// TIA Portal project "EbAndon v2_0_1" (V15)

(* hardware
DEVICE "S71500/ET200MP station_1"  S7-1500 station
   slot 0: "Rail_0"  Rack  6ES7 590-1***0-0AA0
   slot 1: "PLC_1"  CPU 1515F-2 PN  6ES7 515-2FM01-0AB0  V2.5
      slot 3: "CPU display_1"  6ES7591-1BA00-0AA0
DEVICE "HMI_1"  TP1500 Comfort PRO
   slot 0: "HMI_1"  TP1500 Comfort PRO  6AV2 124-0QC24-1AX0  15.0.0.0
   slot 1: "HMI_RT_1"  TP1500 Comfort PRO  6AV2 124-0QC24-1AX0  15.0.0.0
   slot 5: "HMI_1.IE_CP_1"  PROFINET Interface  15.0.0.0
      slot 1: "PROFINET Interface_1"  PROFINET Interface
         slot 1: "Port_1"  Port
         slot 2: "Port_2"  Port
   slot 6: "HMI_1.IE_CP_2"  PROFINET Interface  15.0.0.0
      slot 1: "PROFINET Interface_GBit"  PROFINET Interface
         slot 1: "Port_1"  Port
   slot 7: "HMI_1.MPI/DP_CP_1"  MPI/DP Interface  15.0.0.0
DEVICE "ET 200SP station_1"  ET 200SP-Station
   slot 0: "Rack_0"  Rack  6ES5 710-8MAx1
   slot 0: "station6et200sp"  IM 155-6 PN ST  6ES7 155-6AU01-0BN0  V4.1
   slot 1: "DQ 8x24VDC/0.5A ST_1"  DQ 8x24VDC/0.5A ST  6ES7 132-6BF01-0BA0  V0.0
      slot 1: "DQ 8x24VDC/0.5A ST_1"  DQ 8x24VDC/0.5A ST
   slot 2: "DQ 8x24VDC/0.5A ST_2"  DQ 8x24VDC/0.5A ST  6ES7 132-6BF01-0BA0  V0.0
      slot 1: "DQ 8x24VDC/0.5A ST_2"  DQ 8x24VDC/0.5A ST
   slot 3: "DQ 8x24VDC/0.5A ST_3"  DQ 8x24VDC/0.5A ST  6ES7 132-6BF01-0BA0  V0.0
      slot 1: "DQ 8x24VDC/0.5A ST_3"  DQ 8x24VDC/0.5A ST
   slot 4: "Server module_1"  Server module  6ES7 193-6PA00-0AA0  V1.1
      slot 1: "Server module_1"  Server module
   slot 127: "BA 2xRJ45"  BA 2xRJ45  6ES7 193-6AR00-0AA0  V0.0
      slot 1: "Port_1"  6ES7 193-6AR00-0AA0  V0.0
      slot 2: "Port_2"  6ES7 193-6AR00-0AA0  V0.0
DEVICE "ET 200SP station_2"  ET 200SP-Station
   slot 0: "Rack_0"  Rack  6ES5 710-8MAx1
   slot 0: "station7et200sp"  IM 155-6 PN ST  6ES7 155-6AU01-0BN0  V4.1
   slot 1: "DQ 8x24VDC/0.5A ST_1"  DQ 8x24VDC/0.5A ST  6ES7 132-6BF01-0BA0  V0.0
      slot 1: "DQ 8x24VDC/0.5A ST_1"  DQ 8x24VDC/0.5A ST
   slot 2: "DQ 8x24VDC/0.5A ST_2"  DQ 8x24VDC/0.5A ST  6ES7 132-6BF01-0BA0  V0.0
      slot 1: "DQ 8x24VDC/0.5A ST_2"  DQ 8x24VDC/0.5A ST
   slot 3: "DQ 8x24VDC/0.5A ST_3"  DQ 8x24VDC/0.5A ST  6ES7 132-6BF01-0BA0  V0.0
      slot 1: "DQ 8x24VDC/0.5A ST_3"  DQ 8x24VDC/0.5A ST
   slot 4: "Server module_1"  Server module  6ES7 193-6PA00-0AA0  V1.1
      slot 1: "Server module_1"  Server module
   slot 127: "BA 2xRJ45"  BA 2xRJ45  6ES7 193-6AR00-0AA0  V0.0
      slot 1: "Port_1"  6ES7 193-6AR00-0AA0  V0.0
      slot 2: "Port_2"  6ES7 193-6AR00-0AA0  V0.0
DEVICE "ET 200SP station_3"  ET 200SP-Station
   slot 0: "Rack_0"  Rack  6ES5 710-8MAx1
   slot 0: "station8et200sp"  IM 155-6 PN ST  6ES7 155-6AU01-0BN0  V4.1
   slot 1: "DQ 8x24VDC/0.5A ST_1"  DQ 8x24VDC/0.5A ST  6ES7 132-6BF01-0BA0  V0.0
      slot 1: "DQ 8x24VDC/0.5A ST_1"  DQ 8x24VDC/0.5A ST
   slot 2: "DQ 8x24VDC/0.5A ST_2"  DQ 8x24VDC/0.5A ST  6ES7 132-6BF01-0BA0  V0.0
      slot 1: "DQ 8x24VDC/0.5A ST_2"  DQ 8x24VDC/0.5A ST
   slot 3: "DQ 8x24VDC/0.5A ST_3"  DQ 8x24VDC/0.5A ST  6ES7 132-6BF01-0BA0  V0.0
      slot 1: "DQ 8x24VDC/0.5A ST_3"  DQ 8x24VDC/0.5A ST
   slot 4: "Server module_1"  Server module  6ES7 193-6PA00-0AA0  V1.1
      slot 1: "Server module_1"  Server module
   slot 127: "BA 2xRJ45"  BA 2xRJ45  6ES7 193-6AR00-0AA0  V0.0
      slot 1: "Port_1"  6ES7 193-6AR00-0AA0  V0.0
      slot 2: "Port_2"  6ES7 193-6AR00-0AA0  V0.0
DEVICE "KP8_1"  SIMATIC Key Panel
   slot 0: "Rack"  Rail  V1.0
   slot 0: "station8kp8"  KP8  6AV3 688-3AY36-0AX0  R01.00.00
DEVICE "KP8_2"  SIMATIC Key Panel
   slot 0: "Rack"  Rail  V1.0
   slot 0: "station7kp8"  KP8  6AV3 688-3AY36-0AX0  R01.00.00
DEVICE "KP8_3"  SIMATIC Key Panel
   slot 0: "Rack"  Rail  V1.0
   slot 0: "station6kp8"  KP8  6AV3 688-3AY36-0AX0  R01.00.00
DEVICE "KP8_4"  SIMATIC Key Panel
   slot 0: "Rack"  Rail  V1.0
   slot 0: "station9kp8"  KP8  6AV3 688-3AY36-0AX0  R01.00.00
DEVICE "ET 200SP station_4"  ET 200SP-Station
   slot 0: "Rack_0"  Rack  6ES5 710-8MAx1
   slot 0: "station9et200sp"  IM 155-6 PN ST  6ES7 155-6AU01-0BN0  V4.1
   slot 1: "DQ 8x24VDC/0.5A ST_1"  DQ 8x24VDC/0.5A ST  6ES7 132-6BF01-0BA0  V0.0
      slot 1: "DQ 8x24VDC/0.5A ST_1"  DQ 8x24VDC/0.5A ST
   slot 2: "DQ 8x24VDC/0.5A ST_2"  DQ 8x24VDC/0.5A ST  6ES7 132-6BF01-0BA0  V0.0
      slot 1: "DQ 8x24VDC/0.5A ST_2"  DQ 8x24VDC/0.5A ST
   slot 3: "DQ 8x24VDC/0.5A ST_3"  DQ 8x24VDC/0.5A ST  6ES7 132-6BF01-0BA0  V0.0
      slot 1: "DQ 8x24VDC/0.5A ST_3"  DQ 8x24VDC/0.5A ST
   slot 4: "Server module_1"  Server module  6ES7 193-6PA00-0AA0  V1.1
      slot 1: "Server module_1"  Server module
   slot 127: "BA 2xRJ45"  BA 2xRJ45  6ES7 193-6AR00-0AA0  V0.0
      slot 1: "Port_1"  6ES7 193-6AR00-0AA0  V0.0
      slot 2: "Port_2"  6ES7 193-6AR00-0AA0  V0.0
DEVICE "ET 200SP station_5"  ET 200SP-Station
   slot 0: "Rack_0"  Rack  6ES5 710-8MAx1
   slot 0: "station10et200sp"  IM 155-6 PN ST  6ES7 155-6AU01-0BN0  V4.1
   slot 1: "DQ 8x24VDC/0.5A ST_1"  DQ 8x24VDC/0.5A ST  6ES7 132-6BF01-0BA0  V0.0
      slot 1: "DQ 8x24VDC/0.5A ST_1"  DQ 8x24VDC/0.5A ST
   slot 2: "DQ 8x24VDC/0.5A ST_2"  DQ 8x24VDC/0.5A ST  6ES7 132-6BF01-0BA0  V0.0
      slot 1: "DQ 8x24VDC/0.5A ST_2"  DQ 8x24VDC/0.5A ST
   slot 3: "DQ 8x24VDC/0.5A ST_3"  DQ 8x24VDC/0.5A ST  6ES7 132-6BF01-0BA0  V0.0
      slot 1: "DQ 8x24VDC/0.5A ST_3"  DQ 8x24VDC/0.5A ST
   slot 4: "Server module_1"  Server module  6ES7 193-6PA00-0AA0  V1.1
      slot 1: "Server module_1"  Server module
   slot 127: "BA 2xRJ45"  BA 2xRJ45  6ES7 193-6AR00-0AA0  V0.0
      slot 1: "Port_1"  6ES7 193-6AR00-0AA0  V0.0
      slot 2: "Port_2"  6ES7 193-6AR00-0AA0  V0.0
DEVICE "KP8_5"  SIMATIC Key Panel
   slot 0: "Rack"  Rail  V1.0
   slot 0: "station10kp8"  KP8  6AV3 688-3AY36-0AX0  R01.00.00
DEVICE "KP8_6"  SIMATIC Key Panel
   slot 0: "Rack"  Rail  V1.0
   slot 0: "station11kp8"  KP8  6AV3 688-3AY36-0AX0  R01.00.00
DEVICE "ET 200SP station_6"  ET 200SP-Station
   slot 0: "Rack_0"  Rack  6ES5 710-8MAx1
   slot 0: "station11et200sp"  IM 155-6 PN ST  6ES7 155-6AU01-0BN0  V4.1
   slot 1: "DQ 8x24VDC/0.5A ST_1"  DQ 8x24VDC/0.5A ST  6ES7 132-6BF01-0BA0  V0.0
      slot 1: "DQ 8x24VDC/0.5A ST_1"  DQ 8x24VDC/0.5A ST
   slot 2: "DQ 8x24VDC/0.5A ST_2"  DQ 8x24VDC/0.5A ST  6ES7 132-6BF01-0BA0  V0.0
      slot 1: "DQ 8x24VDC/0.5A ST_2"  DQ 8x24VDC/0.5A ST
   slot 3: "DQ 8x24VDC/0.5A ST_3"  DQ 8x24VDC/0.5A ST  6ES7 132-6BF01-0BA0  V0.0
      slot 1: "DQ 8x24VDC/0.5A ST_3"  DQ 8x24VDC/0.5A ST
   slot 4: "Server module_1"  Server module  6ES7 193-6PA00-0AA0  V1.1
      slot 1: "Server module_1"  Server module
   slot 127: "BA 2xRJ45"  BA 2xRJ45  6ES7 193-6AR00-0AA0  V0.0
      slot 1: "Port_1"  6ES7 193-6AR00-0AA0  V0.0
      slot 2: "Port_2"  6ES7 193-6AR00-0AA0  V0.0
DEVICE "KP8_7"  SIMATIC Key Panel
   slot 0: "Rack"  Rail  V1.0
   slot 0: "station01kp8"  KP8  6AV3 688-3AY36-0AX0  R01.00.00
DEVICE "ET 200SP station_7"  ET 200SP-Station
   slot 0: "Rack_0"  Rack  6ES5 710-8MAx1
   slot 0: "station01et200sp"  IM 155-6 PN ST  6ES7 155-6AU01-0BN0  V4.1
   slot 1: "DQ 8x24VDC/0.5A ST_1"  DQ 8x24VDC/0.5A ST  6ES7 132-6BF01-0BA0  V0.0
      slot 1: "DQ 8x24VDC/0.5A ST_1"  DQ 8x24VDC/0.5A ST
   slot 2: "DQ 8x24VDC/0.5A ST_2"  DQ 8x24VDC/0.5A ST  6ES7 132-6BF01-0BA0  V0.0
      slot 1: "DQ 8x24VDC/0.5A ST_2"  DQ 8x24VDC/0.5A ST
   slot 3: "DQ 8x24VDC/0.5A ST_3"  DQ 8x24VDC/0.5A ST  6ES7 132-6BF01-0BA0  V0.0
      slot 1: "DQ 8x24VDC/0.5A ST_3"  DQ 8x24VDC/0.5A ST
   slot 4: "Server module_1"  Server module  6ES7 193-6PA00-0AA0  V1.1
      slot 1: "Server module_1"  Server module
   slot 127: "BA 2xRJ45"  BA 2xRJ45  6ES7 193-6AR00-0AA0  V0.0
      slot 1: "Port_1"  6ES7 193-6AR00-0AA0  V0.0
      slot 2: "Port_2"  6ES7 193-6AR00-0AA0  V0.0
DEVICE "ET 200SP station_8"  ET 200SP-Station
   slot 0: "Rack_0"  Rack  6ES5 710-8MAx1
   slot 0: "station02et200sp"  IM 155-6 PN ST  6ES7 155-6AU01-0BN0  V4.1
   slot 1: "DQ 8x24VDC/0.5A ST_1"  DQ 8x24VDC/0.5A ST  6ES7 132-6BF01-0BA0  V0.0
      slot 1: "DQ 8x24VDC/0.5A ST_1"  DQ 8x24VDC/0.5A ST
   slot 2: "DQ 8x24VDC/0.5A ST_2"  DQ 8x24VDC/0.5A ST  6ES7 132-6BF01-0BA0  V0.0
      slot 1: "DQ 8x24VDC/0.5A ST_2"  DQ 8x24VDC/0.5A ST
   slot 3: "DQ 8x24VDC/0.5A ST_3"  DQ 8x24VDC/0.5A ST  6ES7 132-6BF01-0BA0  V0.0
      slot 1: "DQ 8x24VDC/0.5A ST_3"  DQ 8x24VDC/0.5A ST
   slot 4: "Server module_1"  Server module  6ES7 193-6PA00-0AA0  V1.1
      slot 1: "Server module_1"  Server module
   slot 127: "BA 2xRJ45"  BA 2xRJ45  6ES7 193-6AR00-0AA0  V0.0
      slot 1: "Port_1"  6ES7 193-6AR00-0AA0  V0.0
      slot 2: "Port_2"  6ES7 193-6AR00-0AA0  V0.0
DEVICE "KP8_8"  SIMATIC Key Panel
   slot 0: "Rack"  Rail  V1.0
   slot 0: "station02kp8"  KP8  6AV3 688-3AY36-0AX0  R01.00.00
DEVICE "KP8_9"  SIMATIC Key Panel
   slot 0: "Rack"  Rail  V1.0
   slot 0: "station03kp8"  KP8  6AV3 688-3AY36-0AX0  R01.00.00
DEVICE "KP8_10"  SIMATIC Key Panel
   slot 0: "Rack"  Rail  V1.0
   slot 0: "station04kp8"  KP8  6AV3 688-3AY36-0AX0  R01.00.00
DEVICE "KP8_11"  SIMATIC Key Panel
   slot 0: "Rack"  Rail  V1.0
   slot 0: "station05kp8"  KP8  6AV3 688-3AY36-0AX0  R01.00.00
DEVICE "ET 200SP station_9"  ET 200SP-Station
   slot 0: "Rack_0"  Rack  6ES5 710-8MAx1
   slot 0: "station03et200sp"  IM 155-6 PN ST  6ES7 155-6AU01-0BN0  V4.1
   slot 1: "DQ 8x24VDC/0.5A ST_1"  DQ 8x24VDC/0.5A ST  6ES7 132-6BF01-0BA0  V0.0
      slot 1: "DQ 8x24VDC/0.5A ST_1"  DQ 8x24VDC/0.5A ST
   slot 2: "DQ 8x24VDC/0.5A ST_2"  DQ 8x24VDC/0.5A ST  6ES7 132-6BF01-0BA0  V0.0
      slot 1: "DQ 8x24VDC/0.5A ST_2"  DQ 8x24VDC/0.5A ST
   slot 3: "DQ 8x24VDC/0.5A ST_3"  DQ 8x24VDC/0.5A ST  6ES7 132-6BF01-0BA0  V0.0
      slot 1: "DQ 8x24VDC/0.5A ST_3"  DQ 8x24VDC/0.5A ST
   slot 4: "Server module_1"  Server module  6ES7 193-6PA00-0AA0  V1.1
      slot 1: "Server module_1"  Server module
   slot 127: "BA 2xRJ45"  BA 2xRJ45  6ES7 193-6AR00-0AA0  V0.0
      slot 1: "Port_1"  6ES7 193-6AR00-0AA0  V0.0
      slot 2: "Port_2"  6ES7 193-6AR00-0AA0  V0.0
DEVICE "ET 200SP station_10"  ET 200SP-Station
   slot 0: "Rack_0"  Rack  6ES5 710-8MAx1
   slot 0: "station04et200sp"  IM 155-6 PN ST  6ES7 155-6AU01-0BN0  V4.1
   slot 1: "DQ 8x24VDC/0.5A ST_1"  DQ 8x24VDC/0.5A ST  6ES7 132-6BF01-0BA0  V0.0
      slot 1: "DQ 8x24VDC/0.5A ST_1"  DQ 8x24VDC/0.5A ST
   slot 2: "DQ 8x24VDC/0.5A ST_2"  DQ 8x24VDC/0.5A ST  6ES7 132-6BF01-0BA0  V0.0
      slot 1: "DQ 8x24VDC/0.5A ST_2"  DQ 8x24VDC/0.5A ST
   slot 3: "DQ 8x24VDC/0.5A ST_3"  DQ 8x24VDC/0.5A ST  6ES7 132-6BF01-0BA0  V0.0
      slot 1: "DQ 8x24VDC/0.5A ST_3"  DQ 8x24VDC/0.5A ST
   slot 4: "Server module_1"  Server module  6ES7 193-6PA00-0AA0  V1.1
      slot 1: "Server module_1"  Server module
   slot 127: "BA 2xRJ45"  BA 2xRJ45  6ES7 193-6AR00-0AA0  V0.0
      slot 1: "Port_1"  6ES7 193-6AR00-0AA0  V0.0
      slot 2: "Port_2"  6ES7 193-6AR00-0AA0  V0.0
DEVICE "ET 200SP station_11"  ET 200SP-Station
   slot 0: "Rack_0"  Rack  6ES5 710-8MAx1
   slot 0: "station05et200sp"  IM 155-6 PN ST  6ES7 155-6AU01-0BN0  V4.1
   slot 1: "DQ 8x24VDC/0.5A ST_1"  DQ 8x24VDC/0.5A ST  6ES7 132-6BF01-0BA0  V0.0
      slot 1: "DQ 8x24VDC/0.5A ST_1"  DQ 8x24VDC/0.5A ST
   slot 2: "DQ 8x24VDC/0.5A ST_2"  DQ 8x24VDC/0.5A ST  6ES7 132-6BF01-0BA0  V0.0
      slot 1: "DQ 8x24VDC/0.5A ST_2"  DQ 8x24VDC/0.5A ST
   slot 3: "DQ 8x24VDC/0.5A ST_3"  DQ 8x24VDC/0.5A ST  6ES7 132-6BF01-0BA0  V0.0
      slot 1: "DQ 8x24VDC/0.5A ST_3"  DQ 8x24VDC/0.5A ST
   slot 4: "Server module_1"  Server module  6ES7 193-6PA00-0AA0  V1.1
      slot 1: "Server module_1"  Server module
   slot 127: "BA 2xRJ45"  BA 2xRJ45  6ES7 193-6AR00-0AA0  V0.0
      slot 1: "Port_1"  6ES7 193-6AR00-0AA0  V0.0
      slot 2: "Port_2"  6ES7 193-6AR00-0AA0  V0.0
DEVICE "PC-System_1"  SIMATIC PC station
   slot 0: "SIMATIC PC station"  Rail  SIMATIC PC-Station  V1.0
      slot 125: "Stationmanager"  Station_Manager  V6.0.4
   slot 1: "HMI_RT_2"  WinCC RT Advanced  6AV2 104-0xxxx-xxxx  15.0.0.0
      slot 33792: "Host interface"  Host interface
   slot 2: "IE general_1"  IE General  IE_CP  V8.2.0
DEVICE "ET 200SP station_12"  ET 200SP-Station
   slot 0: "Rack_0"  Rack  6ES5 710-8MAx1
   slot 0: "chm1et200sp"  IM 155-6 PN ST  6ES7 155-6AU01-0BN0  V4.1
   slot 1: "DQ 8x24VDC/0.5A ST_1"  DQ 8x24VDC/0.5A ST  6ES7 132-6BF01-0BA0  V0.0
      slot 1: "DQ 8x24VDC/0.5A ST_1"  DQ 8x24VDC/0.5A ST
   slot 2: "DQ 8x24VDC/0.5A ST_2"  DQ 8x24VDC/0.5A ST  6ES7 132-6BF01-0BA0  V0.0
      slot 1: "DQ 8x24VDC/0.5A ST_2"  DQ 8x24VDC/0.5A ST
   slot 3: "DQ 8x24VDC/0.5A ST_3"  DQ 8x24VDC/0.5A ST  6ES7 132-6BF01-0BA0  V0.0
      slot 1: "DQ 8x24VDC/0.5A ST_3"  DQ 8x24VDC/0.5A ST
   slot 4: "Server module_1"  Server module  6ES7 193-6PA00-0AA0  V1.1
      slot 1: "Server module_1"  Server module
   slot 127: "BA 2xRJ45"  BA 2xRJ45  6ES7 193-6AR00-0AA0  V0.0
      slot 1: "Port_1"  6ES7 193-6AR00-0AA0  V0.0
      slot 2: "Port_2"  6ES7 193-6AR00-0AA0  V0.0
DEVICE "KP8_12"  SIMATIC Key Panel
   slot 0: "Rack"  Rail  V1.0
   slot 0: "chm1kp8"  KP8  6AV3 688-3AY36-0AX0  R01.00.00
DEVICE "ET 200SP station_13"  ET 200SP-Station
   slot 0: "Rack_0"  Rack  6ES5 710-8MAx1
   slot 0: "chm2et200sp"  IM 155-6 PN ST  6ES7 155-6AU01-0BN0  V4.1
   slot 1: "DQ 8x24VDC/0.5A ST_1"  DQ 8x24VDC/0.5A ST  6ES7 132-6BF01-0BA0  V0.0
      slot 1: "DQ 8x24VDC/0.5A ST_1"  DQ 8x24VDC/0.5A ST
   slot 2: "DQ 8x24VDC/0.5A ST_2"  DQ 8x24VDC/0.5A ST  6ES7 132-6BF01-0BA0  V0.0
      slot 1: "DQ 8x24VDC/0.5A ST_2"  DQ 8x24VDC/0.5A ST
   slot 3: "DQ 8x24VDC/0.5A ST_3"  DQ 8x24VDC/0.5A ST  6ES7 132-6BF01-0BA0  V0.0
      slot 1: "DQ 8x24VDC/0.5A ST_3"  DQ 8x24VDC/0.5A ST
   slot 4: "Server module_1"  Server module  6ES7 193-6PA00-0AA0  V1.1
      slot 1: "Server module_1"  Server module
   slot 127: "BA 2xRJ45"  BA 2xRJ45  6ES7 193-6AR00-0AA0  V0.0
      slot 1: "Port_1"  6ES7 193-6AR00-0AA0  V0.0
      slot 2: "Port_2"  6ES7 193-6AR00-0AA0  V0.0
DEVICE "KP8_13"  SIMATIC Key Panel
   slot 0: "Rack"  Rail  V1.0
   slot 0: "chm2kp8"  KP8  6AV3 688-3AY36-0AX0  R01.00.00
DEVICE "ET 200SP station_14"  ET 200SP-Station
   slot 0: "Rack_0"  Rack  6ES5 710-8MAx1
   slot 0: "chm3et200sp"  IM 155-6 PN ST  6ES7 155-6AU01-0BN0  V4.1
   slot 1: "DQ 8x24VDC/0.5A ST_1"  DQ 8x24VDC/0.5A ST  6ES7 132-6BF01-0BA0  V0.0
      slot 1: "DQ 8x24VDC/0.5A ST_1"  DQ 8x24VDC/0.5A ST
   slot 2: "DQ 8x24VDC/0.5A ST_2"  DQ 8x24VDC/0.5A ST  6ES7 132-6BF01-0BA0  V0.0
      slot 1: "DQ 8x24VDC/0.5A ST_2"  DQ 8x24VDC/0.5A ST
   slot 3: "DQ 8x24VDC/0.5A ST_3"  DQ 8x24VDC/0.5A ST  6ES7 132-6BF01-0BA0  V0.0
      slot 1: "DQ 8x24VDC/0.5A ST_3"  DQ 8x24VDC/0.5A ST
   slot 4: "Server module_1"  Server module  6ES7 193-6PA00-0AA0  V1.1
      slot 1: "Server module_1"  Server module
   slot 127: "BA 2xRJ45"  BA 2xRJ45  6ES7 193-6AR00-0AA0  V0.0
      slot 1: "Port_1"  6ES7 193-6AR00-0AA0  V0.0
      slot 2: "Port_2"  6ES7 193-6AR00-0AA0  V0.0
DEVICE "KP8_14"  SIMATIC Key Panel
   slot 0: "Rack"  Rail  V1.0
   slot 0: "chm3kp8"  KP8  6AV3 688-3AY36-0AX0  R01.00.00
DEVICE "KP8_15"  SIMATIC Key Panel
   slot 0: "Rack"  Rail  V1.0
   slot 0: "chm4kp8"  KP8  6AV3 688-3AY36-0AX0  R01.00.00
DEVICE "ET 200SP station_15"  ET 200SP-Station
   slot 0: "Rack_0"  Rack  6ES5 710-8MAx1
   slot 0: "chm4et200sp"  IM 155-6 PN ST  6ES7 155-6AU01-0BN0  V4.1
   slot 1: "DQ 8x24VDC/0.5A ST_1"  DQ 8x24VDC/0.5A ST  6ES7 132-6BF01-0BA0  V0.0
      slot 1: "DQ 8x24VDC/0.5A ST_1"  DQ 8x24VDC/0.5A ST
   slot 2: "DQ 8x24VDC/0.5A ST_2"  DQ 8x24VDC/0.5A ST  6ES7 132-6BF01-0BA0  V0.0
      slot 1: "DQ 8x24VDC/0.5A ST_2"  DQ 8x24VDC/0.5A ST
   slot 3: "DQ 8x24VDC/0.5A ST_3"  DQ 8x24VDC/0.5A ST  6ES7 132-6BF01-0BA0  V0.0
      slot 1: "DQ 8x24VDC/0.5A ST_3"  DQ 8x24VDC/0.5A ST
   slot 4: "Server module_1"  Server module  6ES7 193-6PA00-0AA0  V1.1
      slot 1: "Server module_1"  Server module
   slot 127: "BA 2xRJ45"  BA 2xRJ45  6ES7 193-6AR00-0AA0  V0.0
      slot 1: "Port_1"  6ES7 193-6AR00-0AA0  V0.0
      slot 2: "Port_2"  6ES7 193-6AR00-0AA0  V0.0
DEVICE "KP8_16"  SIMATIC Key Panel
   slot 0: "Rack"  Rail  V1.0
   slot 0: "cdo1kp8"  KP8  6AV3 688-3AY36-0AX0  R01.00.00
DEVICE "ET 200SP station_16"  ET 200SP-Station
   slot 0: "Rack_0"  Rack  6ES5 710-8MAx1
   slot 0: "cdo1et200sp"  IM 155-6 PN ST  6ES7 155-6AU01-0BN0  V4.1
   slot 1: "DQ 8x24VDC/0.5A ST_1"  DQ 8x24VDC/0.5A ST  6ES7 132-6BF01-0BA0  V0.0
      slot 1: "DQ 8x24VDC/0.5A ST_1"  DQ 8x24VDC/0.5A ST
   slot 2: "DQ 8x24VDC/0.5A ST_2"  DQ 8x24VDC/0.5A ST  6ES7 132-6BF01-0BA0  V0.0
      slot 1: "DQ 8x24VDC/0.5A ST_2"  DQ 8x24VDC/0.5A ST
   slot 3: "DQ 8x24VDC/0.5A ST_3"  DQ 8x24VDC/0.5A ST  6ES7 132-6BF01-0BA0  V0.0
      slot 1: "DQ 8x24VDC/0.5A ST_3"  DQ 8x24VDC/0.5A ST
   slot 4: "Server module_1"  Server module  6ES7 193-6PA00-0AA0  V1.1
      slot 1: "Server module_1"  Server module
   slot 127: "BA 2xRJ45"  BA 2xRJ45  6ES7 193-6AR00-0AA0  V0.0
      slot 1: "Port_1"  6ES7 193-6AR00-0AA0  V0.0
      slot 2: "Port_2"  6ES7 193-6AR00-0AA0  V0.0
DEVICE "ET 200SP station_17"  ET 200SP-Station
   slot 0: "Rack_0"  Rack  6ES5 710-8MAx1
   slot 0: "cdo2et200sp"  IM 155-6 PN ST  6ES7 155-6AU01-0BN0  V4.1
   slot 1: "DQ 8x24VDC/0.5A ST_1"  DQ 8x24VDC/0.5A ST  6ES7 132-6BF01-0BA0  V0.0
      slot 1: "DQ 8x24VDC/0.5A ST_1"  DQ 8x24VDC/0.5A ST
   slot 2: "DQ 8x24VDC/0.5A ST_2"  DQ 8x24VDC/0.5A ST  6ES7 132-6BF01-0BA0  V0.0
      slot 1: "DQ 8x24VDC/0.5A ST_2"  DQ 8x24VDC/0.5A ST
   slot 3: "DQ 8x24VDC/0.5A ST_3"  DQ 8x24VDC/0.5A ST  6ES7 132-6BF01-0BA0  V0.0
      slot 1: "DQ 8x24VDC/0.5A ST_3"  DQ 8x24VDC/0.5A ST
   slot 4: "Server module_1"  Server module  6ES7 193-6PA00-0AA0  V1.1
      slot 1: "Server module_1"  Server module
   slot 127: "BA 2xRJ45"  BA 2xRJ45  6ES7 193-6AR00-0AA0  V0.0
      slot 1: "Port_1"  6ES7 193-6AR00-0AA0  V0.0
      slot 2: "Port_2"  6ES7 193-6AR00-0AA0  V0.0
DEVICE "KP8_17"  SIMATIC Key Panel
   slot 0: "Rack"  Rail  V1.0
   slot 0: "cdo2kp8"  KP8  6AV3 688-3AY36-0AX0  R01.00.00
DEVICE "KP8_18"  SIMATIC Key Panel
   slot 0: "Rack"  Rail  V1.0
   slot 0: "cdo3kp8"  KP8  6AV3 688-3AY36-0AX0  R01.00.00
DEVICE "ET 200SP station_18"  ET 200SP-Station
   slot 0: "Rack_0"  Rack  6ES5 710-8MAx1
   slot 0: "cdo3et200sp"  IM 155-6 PN ST  6ES7 155-6AU01-0BN0  V4.1
   slot 1: "DQ 8x24VDC/0.5A ST_1"  DQ 8x24VDC/0.5A ST  6ES7 132-6BF01-0BA0  V0.0
      slot 1: "DQ 8x24VDC/0.5A ST_1"  DQ 8x24VDC/0.5A ST
   slot 2: "DQ 8x24VDC/0.5A ST_2"  DQ 8x24VDC/0.5A ST  6ES7 132-6BF01-0BA0  V0.0
      slot 1: "DQ 8x24VDC/0.5A ST_2"  DQ 8x24VDC/0.5A ST
   slot 3: "DQ 8x24VDC/0.5A ST_3"  DQ 8x24VDC/0.5A ST  6ES7 132-6BF01-0BA0  V0.0
      slot 1: "DQ 8x24VDC/0.5A ST_3"  DQ 8x24VDC/0.5A ST
   slot 4: "Server module_1"  Server module  6ES7 193-6PA00-0AA0  V1.1
      slot 1: "Server module_1"  Server module
   slot 127: "BA 2xRJ45"  BA 2xRJ45  6ES7 193-6AR00-0AA0  V0.0
      slot 1: "Port_1"  6ES7 193-6AR00-0AA0  V0.0
      slot 2: "Port_2"  6ES7 193-6AR00-0AA0  V0.0
DEVICE "ET 200SP station_19"  ET 200SP-Station
   slot 0: "Rack_0"  Rack  6ES5 710-8MAx1
   slot 0: "bfl1et200sp"  IM 155-6 PN ST  6ES7 155-6AU01-0BN0  V4.1
   slot 1: "DQ 8x24VDC/0.5A ST_1"  DQ 8x24VDC/0.5A ST  6ES7 132-6BF01-0BA0  V0.0
      slot 1: "DQ 8x24VDC/0.5A ST_1"  DQ 8x24VDC/0.5A ST
   slot 2: "DQ 8x24VDC/0.5A ST_2"  DQ 8x24VDC/0.5A ST  6ES7 132-6BF01-0BA0  V0.0
      slot 1: "DQ 8x24VDC/0.5A ST_2"  DQ 8x24VDC/0.5A ST
   slot 3: "DQ 8x24VDC/0.5A ST_3"  DQ 8x24VDC/0.5A ST  6ES7 132-6BF01-0BA0  V0.0
      slot 1: "DQ 8x24VDC/0.5A ST_3"  DQ 8x24VDC/0.5A ST
   slot 4: "Server module_1"  Server module  6ES7 193-6PA00-0AA0  V1.1
      slot 1: "Server module_1"  Server module
   slot 127: "BA 2xRJ45"  BA 2xRJ45  6ES7 193-6AR00-0AA0  V0.0
      slot 1: "Port_1"  6ES7 193-6AR00-0AA0  V0.0
      slot 2: "Port_2"  6ES7 193-6AR00-0AA0  V0.0
DEVICE "KP8_19"  SIMATIC Key Panel
   slot 0: "Rack"  Rail  V1.0
   slot 0: "bfl1kp8"  KP8  6AV3 688-3AY36-0AX0  R01.00.00
DEVICE "KP8_20"  SIMATIC Key Panel
   slot 0: "Rack"  Rail  V1.0
   slot 0: "bfl2kp8"  KP8  6AV3 688-3AY36-0AX0  R01.00.00
DEVICE "ET 200SP station_20"  ET 200SP-Station
   slot 0: "Rack_0"  Rack  6ES5 710-8MAx1
   slot 0: "bfl2et200sp"  IM 155-6 PN ST  6ES7 155-6AU01-0BN0  V4.1
   slot 1: "DQ 8x24VDC/0.5A ST_1"  DQ 8x24VDC/0.5A ST  6ES7 132-6BF01-0BA0  V0.0
      slot 1: "DQ 8x24VDC/0.5A ST_1"  DQ 8x24VDC/0.5A ST
   slot 2: "DQ 8x24VDC/0.5A ST_2"  DQ 8x24VDC/0.5A ST  6ES7 132-6BF01-0BA0  V0.0
      slot 1: "DQ 8x24VDC/0.5A ST_2"  DQ 8x24VDC/0.5A ST
   slot 3: "DQ 8x24VDC/0.5A ST_3"  DQ 8x24VDC/0.5A ST  6ES7 132-6BF01-0BA0  V0.0
      slot 1: "DQ 8x24VDC/0.5A ST_3"  DQ 8x24VDC/0.5A ST
   slot 4: "Server module_1"  Server module  6ES7 193-6PA00-0AA0  V1.1
      slot 1: "Server module_1"  Server module
   slot 127: "BA 2xRJ45"  BA 2xRJ45  6ES7 193-6AR00-0AA0  V0.0
      slot 1: "Port_1"  6ES7 193-6AR00-0AA0  V0.0
      slot 2: "Port_2"  6ES7 193-6AR00-0AA0  V0.0
DEVICE "ET 200SP station_21"  ET 200SP-Station
   slot 0: "Rack_0"  Rack  6ES5 710-8MAx1
   slot 0: "bfl3et200sp"  IM 155-6 PN ST  6ES7 155-6AU01-0BN0  V4.1
   slot 1: "DQ 8x24VDC/0.5A ST_1"  DQ 8x24VDC/0.5A ST  6ES7 132-6BF01-0BA0  V0.0
      slot 1: "DQ 8x24VDC/0.5A ST_1"  DQ 8x24VDC/0.5A ST
   slot 2: "DQ 8x24VDC/0.5A ST_2"  DQ 8x24VDC/0.5A ST  6ES7 132-6BF01-0BA0  V0.0
      slot 1: "DQ 8x24VDC/0.5A ST_2"  DQ 8x24VDC/0.5A ST
   slot 3: "DQ 8x24VDC/0.5A ST_3"  DQ 8x24VDC/0.5A ST  6ES7 132-6BF01-0BA0  V0.0
      slot 1: "DQ 8x24VDC/0.5A ST_3"  DQ 8x24VDC/0.5A ST
   slot 4: "Server module_1"  Server module  6ES7 193-6PA00-0AA0  V1.1
      slot 1: "Server module_1"  Server module
   slot 127: "BA 2xRJ45"  BA 2xRJ45  6ES7 193-6AR00-0AA0  V0.0
      slot 1: "Port_1"  6ES7 193-6AR00-0AA0  V0.0
      slot 2: "Port_2"  6ES7 193-6AR00-0AA0  V0.0
DEVICE "KP8_21"  SIMATIC Key Panel
   slot 0: "Rack"  Rail  V1.0
   slot 0: "bfl3kp8"  KP8  6AV3 688-3AY36-0AX0  R01.00.00
DEVICE "KP8_22"  SIMATIC Key Panel
   slot 0: "Rack"  Rail  V1.0
   slot 0: "lgs1kp8"  KP8  6AV3 688-3AY36-0AX0  R01.00.00
DEVICE "ET 200SP station_22"  ET 200SP-Station
   slot 0: "Rack_0"  Rack  6ES5 710-8MAx1
   slot 0: "lgs1et200sp"  IM 155-6 PN ST  6ES7 155-6AU01-0BN0  V4.1
   slot 1: "DQ 8x24VDC/0.5A ST_1"  DQ 8x24VDC/0.5A ST  6ES7 132-6BF01-0BA0  V0.0
      slot 1: "DQ 8x24VDC/0.5A ST_1"  DQ 8x24VDC/0.5A ST
   slot 2: "DQ 8x24VDC/0.5A ST_2"  DQ 8x24VDC/0.5A ST  6ES7 132-6BF01-0BA0  V0.0
      slot 1: "DQ 8x24VDC/0.5A ST_2"  DQ 8x24VDC/0.5A ST
   slot 3: "DQ 8x24VDC/0.5A ST_3"  DQ 8x24VDC/0.5A ST  6ES7 132-6BF01-0BA0  V0.0
      slot 1: "DQ 8x24VDC/0.5A ST_3"  DQ 8x24VDC/0.5A ST
   slot 4: "Server module_1"  Server module  6ES7 193-6PA00-0AA0  V1.1
      slot 1: "Server module_1"  Server module
   slot 127: "BA 2xRJ45"  BA 2xRJ45  6ES7 193-6AR00-0AA0  V0.0
      slot 1: "Port_1"  6ES7 193-6AR00-0AA0  V0.0
      slot 2: "Port_2"  6ES7 193-6AR00-0AA0  V0.0
DEVICE "ET 200SP station_23"  ET 200SP-Station
   slot 0: "Rack_0"  Rack  6ES5 710-8MAx1
   slot 0: "lgs2et200sp"  IM 155-6 PN ST  6ES7 155-6AU01-0BN0  V4.1
   slot 1: "DQ 8x24VDC/0.5A ST_1"  DQ 8x24VDC/0.5A ST  6ES7 132-6BF01-0BA0  V0.0
      slot 1: "DQ 8x24VDC/0.5A ST_1"  DQ 8x24VDC/0.5A ST
   slot 2: "DQ 8x24VDC/0.5A ST_2"  DQ 8x24VDC/0.5A ST  6ES7 132-6BF01-0BA0  V0.0
      slot 1: "DQ 8x24VDC/0.5A ST_2"  DQ 8x24VDC/0.5A ST
   slot 3: "DQ 8x24VDC/0.5A ST_3"  DQ 8x24VDC/0.5A ST  6ES7 132-6BF01-0BA0  V0.0
      slot 1: "DQ 8x24VDC/0.5A ST_3"  DQ 8x24VDC/0.5A ST
   slot 4: "Server module_1"  Server module  6ES7 193-6PA00-0AA0  V1.1
      slot 1: "Server module_1"  Server module
   slot 127: "BA 2xRJ45"  BA 2xRJ45  6ES7 193-6AR00-0AA0  V0.0
      slot 1: "Port_1"  6ES7 193-6AR00-0AA0  V0.0
      slot 2: "Port_2"  6ES7 193-6AR00-0AA0  V0.0
DEVICE "KP8_23"  SIMATIC Key Panel
   slot 0: "Rack"  Rail  V1.0
   slot 0: "lgs2kp8"  KP8  6AV3 688-3AY36-0AX0  R01.00.00
*)

// ===== PLC "PLC_1"  CPU 1515F-2 PN =====

VAR_GLOBAL   // PLC tag table "Default tag table"
   "System_Byte" AT %MB1 : Byte;
   "FirstScan" AT %M1.0 : Bool;
   "DiagStatusUpdate" AT %M1.1 : Bool;
   "AlwaysTRUE" AT %M1.2 : Bool;
   "AlwaysFALSE" AT %M1.3 : Bool;
   "Clock_Byte" AT %MB0 : Byte;
   "Clock_10Hz" AT %M0.0 : Bool;
   "Clock_5Hz" AT %M0.1 : Bool;
   "Clock_2.5Hz" AT %M0.2 : Bool;
   "Clock_2Hz" AT %M0.3 : Bool;
   "Clock_1.25Hz" AT %M0.4 : Bool;
   "Clock_1Hz" AT %M0.5 : Bool;
   "Clock_0.625Hz" AT %M0.6 : Bool;
   "Clock_0.5Hz" AT %M0.7 : Bool;
   "Temp Reset" AT %M2.0 : Bool;
END_VAR

VAR_GLOBAL   // PLC tag table "VOLVO 16 1"
   "VOLVO 16 1 IO" AT %QD100 : DWord;
   "VOLVO 16 1 KP8 In" AT %ID0 : DWord;
   "VOLVO 16 1 KP8 Out" AT %QD0 : DWord;
END_VAR

VAR_GLOBAL   // PLC tag table "VOLVO 16 2"
   "VOLVO 16 2 IO" AT %QD104 : DWord;
   "VOLVO 16 2 KP8 In" AT %ID4 : DWord;
   "VOLVO 16 2 KP8 Out" AT %QD4 : DWord;
END_VAR

VAR_GLOBAL   // PLC tag table "VOLVO 16 3"
   "VOLVO 16 3 IO" AT %QD108 : DWord;
   "VOLVO 16 3 KP8 In" AT %ID8 : DWord;
   "VOLVO 16 3 KP8 Out" AT %QD8 : DWord;
END_VAR

VAR_GLOBAL   // PLC tag table "VOLVO 16 4"
   "VOLVO 16 4 IO" AT %QD112 : DWord;
   "VOLVO 16 4 KP8 In" AT %ID12 : DWord;
   "VOLVO 16 4 KP8 Out" AT %QD12 : DWord;
END_VAR

VAR_GLOBAL   // PLC tag table "VOLVO 16 5"
   "VOLVO 16 5 IO" AT %QD116 : DWord;
   "VOLVO 16 5 KP8 In" AT %ID16 : DWord;
   "VOLVO 16 5 KP8 Out" AT %QD16 : DWord;
END_VAR

VAR_GLOBAL   // PLC tag table "VOLVO 16 6"
   "VOLVO 16 6 IO" AT %QD120 : DWord;
   "VOLVO 16 6 KP8 In" AT %ID20 : DWord;
   "VOLVO 16 6 KP8 Out" AT %QD20 : DWord;
END_VAR

VAR_GLOBAL   // PLC tag table "VOLVO 16 7"
   "VOLVO 16 7 IO" AT %QD124 : DWord;
   "VOLVO 16 7 KP8 In" AT %ID24 : DWord;
   "VOLVO 16 7 KP8 Out" AT %QD24 : DWord;
END_VAR

VAR_GLOBAL   // PLC tag table "VOLVO 16 8"
   "VOLVO 16 8 IO" AT %QD128 : DWord;
   "VOLVO 16 8 KP8 In" AT %ID28 : DWord;
   "VOLVO 16 8 KP8 Out" AT %QD28 : DWord;
END_VAR

VAR_GLOBAL   // PLC tag table "VOLVO 16 9"
   "VOLVO 16 9 IO" AT %QD132 : DWord;
   "VOLVO 16 9 KP8 In" AT %ID32 : DWord;
   "VOLVO 16 9 KP8 Out" AT %QD32 : DWord;
END_VAR

VAR_GLOBAL   // PLC tag table "VOLVO 16 10"
   "VOLVO 16 10 IO" AT %QD136 : DWord;
   "VOLVO 16 10 KP8 In" AT %ID36 : DWord;
   "VOLVO 16 10 KP8 Out" AT %QD36 : DWord;
END_VAR

VAR_GLOBAL   // PLC tag table "VOLVO 16 11"
   "VOLVO 16 11 IO" AT %QD140 : DWord;
   "VOLVO 16 11 KP8 In" AT %ID40 : DWord;
   "VOLVO 16 11 KP8 Out" AT %QD40 : DWord;
END_VAR

VAR_GLOBAL   // PLC tag table "CHM 01"
   "CHM 1 KP8 In" AT %ID44 : DWord;
   "CHM 1 KP8 Out" AT %QD44 : DWord;
   "CHM 1 IO" AT %QD144 : DWord;
END_VAR

VAR_GLOBAL   // PLC tag table "CHM 02"
   "CHM 2 IO" AT %QD148 : DWord;
   "CHM 2 KP8 In" AT %ID48 : DWord;
   "CHM 2 KP8 Out" AT %QD48 : DWord;
END_VAR

VAR_GLOBAL   // PLC tag table "CHM 03"
   "CHM 3 IO" AT %QD152 : DWord;
   "CHM 3 KP8 In" AT %ID52 : DWord;
   "CHM 3 KP8 Out" AT %QD52 : DWord;
END_VAR

VAR_GLOBAL   // PLC tag table "CHM 04"
   "CHM 4 IO" AT %QD156 : DWord;
   "CHM 4 KP8 In" AT %ID56 : DWord;
   "CHM 4 KP8 Out" AT %QD56 : DWord;
END_VAR

VAR_GLOBAL   // PLC tag table "CDO 01"
   "CDO 1 IO" AT %QD160 : DWord;
   "CDO 1 KP8 In" AT %ID60 : DWord;
   "CDO 1 KP8 Out" AT %QD60 : DWord;
END_VAR

VAR_GLOBAL   // PLC tag table "CDO 02"
   "CDO 2 IO" AT %QD164 : DWord;
   "CDO 2 KP8 In" AT %ID64 : DWord;
   "CDO 2 KP8 Out" AT %QD64 : DWord;
END_VAR

VAR_GLOBAL   // PLC tag table "CDO 03"
   "CDO 3 IO" AT %QD168 : DWord;
   "CDO 3 KP8 In" AT %ID68 : DWord;
   "CDO 3 KP8 Out" AT %QD68 : DWord;
END_VAR

VAR_GLOBAL   // PLC tag table "BFL 01"
   "BFL 1 IO" AT %QD172 : DWord;
   "BFL 1 KP8 In" AT %ID72 : DWord;
   "BFL 1 KP8 Out" AT %QD72 : DWord;
END_VAR

VAR_GLOBAL   // PLC tag table "BFL 02"
   "BFL 2 IO" AT %QD176 : DWord;
   "BFL 2 KP8 In" AT %ID76 : DWord;
   "BFL 2 KP8 Out" AT %QD76 : DWord;
END_VAR

VAR_GLOBAL   // PLC tag table "BFL 03"
   "BFL 3 IO" AT %QD180 : DWord;
   "BFL 3 KP8 In" AT %ID80 : DWord;
   "BFL 3 KP8 Out" AT %QD80 : DWord;
END_VAR

VAR_GLOBAL   // PLC tag table "LGS 01"
   "LGS 1 IO" AT %QD184 : DWord;
   "LGS 1 KP8 In" AT %ID84 : DWord;
   "LGS 1 KP8 Out" AT %QD84 : DWord;
END_VAR

VAR_GLOBAL   // PLC tag table "LGS 02"
   "LGS 2 IO" AT %QD188 : DWord;
   "LGS 2 KP8 In" AT %ID88 : DWord;
   "LGS 2 KP8 Out" AT %QD88 : DWord;
END_VAR

TYPE "Stations"
   STRUCT
      current : Array[0..22] of "Station";
      old : Array[0..22] of "Station";
   END_STRUCT;
END_TYPE

TYPE "Part Call Screen"
   STRUCT
      current : Array[0..10] of "Table Row";
      old : Array[0..10] of "Table Row";
   END_STRUCT;
END_TYPE

TYPE "Settings Screen"
   STRUCT
      current : "Settings";
      old : "Settings";
   END_STRUCT;
END_TYPE

TYPE "Barcode Screen"
   STRUCT
      partNumber : WString[40];
      barcode : String;
      orderCancelled : Bool;
      ordered : Bool;
   END_STRUCT;
END_TYPE

TYPE "Table Row"
   STRUCT
      address : UInt;
      ordered : Bool;
      pbSelection : Struct
         request : Bool;
         visibility : Bool;
      END_STRUCT;
      rtBackground : Struct
         animatior : UInt;
         visibility : Bool;
      END_STRUCT;
      selected : Bool;
      tfDropZone : Struct
         value : WString[20];
         animator : UInt;
         visibility : Bool;
      END_STRUCT;
      tfLine : Struct
         value : WString[20];
         animator : UInt;
         visibility : Bool;
      END_STRUCT;
      tfPartNumber : Struct
         value : WString[40];
         animator : UInt;
         visibility : Bool;
      END_STRUCT;
      tfTime : Struct
         value : WString[20];
         animator : UInt;
         visibility : Bool;
      END_STRUCT;
   END_STRUCT;
END_TYPE

TYPE "Runtime Data"
   STRUCT
      asReal : Real;
      elapsed : LReal;
      mem : LReal;
   END_STRUCT;
END_TYPE

TYPE "KP8 Button Config"
   STRUCT
      activate : Array[0..7] of Bool;
      colorOn1 : Array[0..7] of String[10];
      colorOn2 : Array[0..7] of String[10];
      colorOff : Array[0..7] of String[10];
      flash : Array[0..7] of Bool;
      group : Array[0..7] of Int;
      mode : Array[0..7] of Bool;
   END_STRUCT;
END_TYPE

TYPE "Constants"
   STRUCT
      buttonCount : Int := 6;   // max buttons per station
      hmiRowCount : Int := 11;   // number of rows displayed on hmi
      stationCount : Int := 23;   // total number of stations
      stationLabelCount : Int := 12;   // labels for settings screen
      partReqRows : Int := 200;
   END_STRUCT;
END_TYPE

TYPE "Part Request Data"
   STRUCT
      row : Array[0..199] of "Table Row";
   END_STRUCT;
END_TYPE

TYPE "Station"
   STRUCT
      animations : Array[0..7] of Int;
      btnStates : Array[0..7] of Bool;
      dropZone : USInt;
      elapsedTime : Struct
         partReq : Array[0..7] of Real;
         resetReq : Real;
      END_STRUCT;
      kp8Config : "KP8 Button Config";
      kp8In : Byte;
      kp8Out : DWord;
      init : Struct
         hard : Bool;
         soft : Bool;
      END_STRUCT;
      line : WString[20];
      partNumbers : Array[0..7] of WString[40];
      partOrdered : Array[0..7] of Bool;
      presetTime : Struct
         allotted : Array[0..7] of Real;
         critical : Array[0..7] of Real;
      END_STRUCT;
      stackLightOut : DWord;
      settings : Struct
         selected : Bool;
         btnSelection : Array[0..7] of Bool;
      END_STRUCT;
   END_STRUCT;
END_TYPE

TYPE "Settings"
   STRUCT
      alotted : Struct
         enable : Bool;
         setTimer : Bool;
         value : WString[10];
      END_STRUCT;
      critical : Struct
         enable : Bool;
         setTimer : Bool;
         value : WString[10];
      END_STRUCT;
      kp8 : Struct
         assign : "Push Button";
         buttons : Array[0..5] of Struct
            animation : Int;
            select : Bool;
            selState : Bool;
         END_STRUCT;
         selCount : Int;
      END_STRUCT;
      stations : Struct
         assign : Struct
            act : Bool;
            enable : Bool;
         END_STRUCT;
         buttons : Array[0..11] of Struct
            label : WString [20];
            select : Bool;
         END_STRUCT;
         nextGroup : Struct
            act : Bool;
            ani : Int;
            enable : Bool;
         END_STRUCT;
         prevGroup : Struct
            act : Bool;
            ani : Int;
            enable : Bool;
         END_STRUCT;
         selCount : Int;
         selState : Array[0..11] of Bool;
      END_STRUCT;
      partNumber : Struct
         enable : Bool;
         enter : Bool;
         value : WString [40];
      END_STRUCT;
      viewingStation : Struct
         btns : Array[0..5] of Struct
            alloted : WString[10];
            critical : WString[10];
            partNumber : WString[40];
         END_STRUCT;
         dzValue : Int;
         lineValue : WString[10];
         next : "Push Button";
         number : Int;
         previous : "Push Button";
         "name" : WString[10];
      END_STRUCT;
   END_STRUCT;
END_TYPE

TYPE "Push Button"
   STRUCT
      act : Bool;
      ani : Int;
      enable : Bool;
   END_STRUCT;
END_TYPE

DATA_BLOCK "EMP IDB"   // DB1
{ S7_Optimized_Access := 'TRUE' }
VERSION : 0.1
// stored: InstanceOfName EMP
"EMP"
BEGIN
   constants.buttonCount := 8;
   stations.current[0].presetTime.allotted[7] := 1800.0;
   stations.current[0].presetTime.allotted[6] := 1800.0;
   stations.current[0].presetTime.allotted[5] := 1800.0;
   stations.current[0].presetTime.allotted[3] := 1800.0;
   stations.current[0].presetTime.allotted[2] := 1800.0;
   stations.current[0].presetTime.allotted[1] := 1800.0;
   stations.current[0].presetTime.critical[7] := 300.0;
   stations.current[0].presetTime.critical[6] := 300.0;
   stations.current[0].presetTime.critical[5] := 300.0;
   stations.current[0].presetTime.critical[3] := 300.0;
   stations.current[0].presetTime.critical[2] := 300.0;
   stations.current[0].presetTime.critical[1] := 300.0;
   stations.current[0].partNumbers[7] := WSTRING#'S1P1';
   stations.current[0].partNumbers[6] := WSTRING#'S1P3';
   stations.current[0].partNumbers[5] := WSTRING#'S1P5';
   stations.current[0].partNumbers[3] := WSTRING#'S1P2';
   stations.current[0].partNumbers[2] := WSTRING#'S1P4';
   stations.current[0].partNumbers[1] := WSTRING#'S1P6';
   stations.current[0].line := WSTRING#'VOLVO 16';
   stations.current[1].line := WSTRING#'VOLVO 16';
   stations.current[2].line := WSTRING#'VOLVO 16';
END_DATA_BLOCK

DATA_BLOCK "HMI"   // DB2
{ S7_Optimized_Access := 'TRUE' }
VERSION : 0.1
   VAR
      partCall : "Part Call Screen";
      screenNumber : Int;
      settings : "Settings Screen";
      barcode : "Barcode Screen";
   END_VAR
BEGIN
END_DATA_BLOCK

DATA_BLOCK "Parts"   // DB3
{ S7_Optimized_Access := 'TRUE' }
VERSION : 0.1
   VAR
      pRow : Int;
   END_VAR
   VAR RETAIN
      requests : "Part Request Data";
   END_VAR
BEGIN
END_DATA_BLOCK

FUNCTION_BLOCK "EMP"   // FB1, LAD
{ S7_Optimized_Access := 'TRUE' }
VERSION : 0.1
   VAR RETAIN
      constants : "Constants";
   END_VAR
   VAR
      instBaseAnimations : "Base Animations";
      instHMIAnimations : "HMI Part Call Animations";
      instInitialize : "Initialize";
      instKP8ButtonActivation : "KP8 Button Activation";
      instKP8ExpandedAnimations : "KP8 Expanded Animations";
      instPartTimers : "Part Timers";
      instRecordPartRequest : "Record Part Request";
      instRemovePartRequest : "Remove Part Request";
      instResetInitRequest : "Reset Init Requests";
      instStackLightAnimations : "Stack Light Animations";
      "KP8 Drivers" : Array[0..#stationCount] of "KP8 Driver";
   END_VAR
   VAR RETAIN
      stations : "Stations";
   END_VAR
   VAR
      instHMIBarcode : "HMI Barcod Screen";
      instCollapseTable : "Collapse Table";
      instPopulateHMI : "HMI Populate Part Call";
      instHMISettings : "HMI Settings Screen";
   END_VAR
   VAR_TEMP
      i : Int;
   END_VAR
   VAR CONSTANT
      stationCount : Int := 22;
   END_VAR
BEGIN

REGION Network 1: PHYSICAL TO GLOBAL
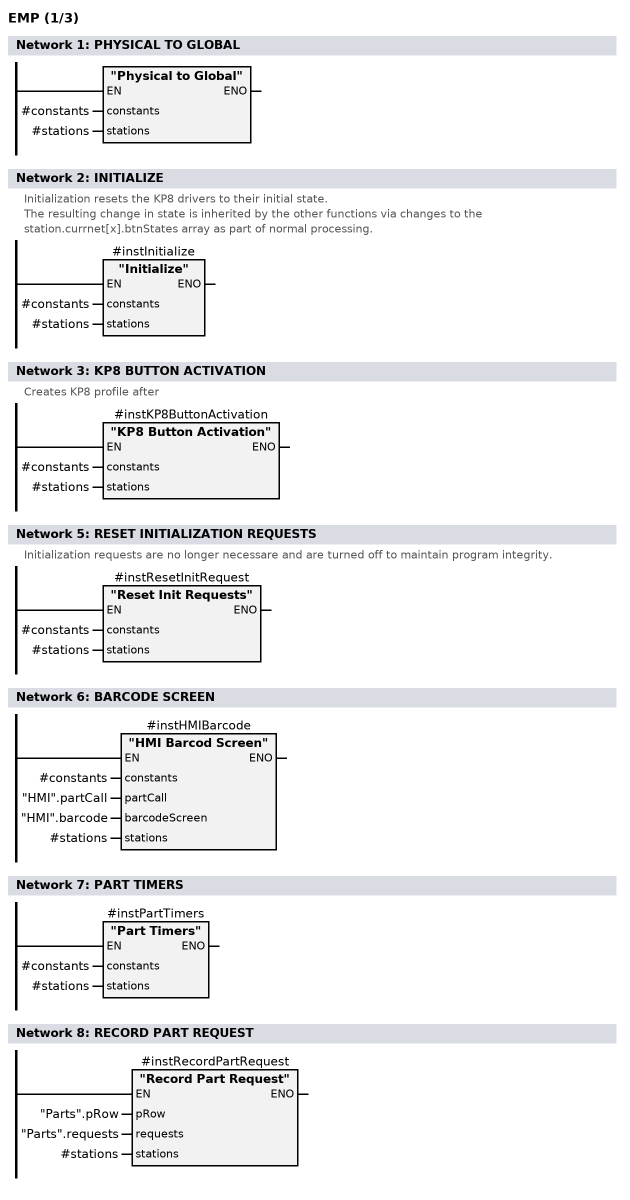
   RUNG wire#powerrail
      "Physical to Global"(constants := #constants, stations := #stations)
   END_RUNG
   // the same network as SCL:
   "Physical to Global"(constants := #constants, stations := #stations);
END_REGION

REGION Network 2: INITIALIZE
   // Initialization resets the KP8 drivers to their initial state.
   // The resulting change in state is inherited by the other functions via changes to the
   // station.currnet[x].btnStates array as part of normal processing.
   RUNG wire#powerrail
      #instInitialize(constants := #constants, stations := #stations)
   END_RUNG
   // the same network as SCL:
   #instInitialize(constants := #constants, stations := #stations);   // "Initialize"
END_REGION

REGION Network 3: KP8 BUTTON ACTIVATION
   // Creates KP8 profile after
   RUNG wire#powerrail
      #instKP8ButtonActivation(constants := #constants, stations := #stations)
   END_RUNG
   // the same network as SCL:
   #instKP8ButtonActivation(constants := #constants, stations := #stations);   // "KP8 Button Activation"
END_REGION

REGION Network 4 (SCL): KP8 DRIVER CALLS
   REGION "LOOP THROUGH STATIONS"
       FOR #i := 0 TO #stationCount DO
           #"KP8 Drivers"[#i](btnIn := #stations.current[#i].kp8In,
                              hardInit := #stations.current[#i].init.hard,
                              softInit := #stations.current[#i].init.soft,
                              btn0Activate := #stations.current[#i].kp8Config.activate[0],
                              btn0Mode := #stations.current[#i].kp8Config.mode[0],
                              btn0Group := #stations.current[#i].kp8Config.group[0],
                              btn0Flash := #stations.current[#i].kp8Config.flash[0],
                              btn0ColorOn1 := #stations.current[#i].kp8Config.colorOn1[0],
                              btn0ColorOn2 := #stations.current[#i].kp8Config.colorOn2[0],
                              btn0ColorOff := #stations.current[#i].kp8Config.colorOff[0],
                              btn1Activate := #stations.current[#i].kp8Config.activate[1],
                              btn1Mode := #stations.current[#i].kp8Config.mode[1],
                              btn1Group := #stations.current[#i].kp8Config.group[1],
                              btn1Flash := #stations.current[#i].kp8Config.flash[1],
                              btn1ColorOn1 := #stations.current[#i].kp8Config.colorOn1[1],
                              btn1ColorOn2 := #stations.current[#i].kp8Config.colorOn2[1],
                              btn1ColorOff := #stations.current[#i].kp8Config.colorOff[1],
                              btn2Activate := #stations.current[#i].kp8Config.activate[2],
                              btn2Mode := #stations.current[#i].kp8Config.mode[2],
                              btn2Group := #stations.current[#i].kp8Config.group[2],
                              btn2Flash := #stations.current[#i].kp8Config.flash[2],
                              btn2ColorOn1 := #stations.current[#i].kp8Config.colorOn1[2],
                              btn2ColorOn2 := #stations.current[#i].kp8Config.colorOn2[2],
                              btn2ColorOff := #stations.current[#i].kp8Config.colorOff[2],
                              btn3Activate := #stations.current[#i].kp8Config.activate[3],
                              btn3Mode := #stations.current[#i].kp8Config.mode[3],
                              btn3Group := #stations.current[#i].kp8Config.group[3],
                              btn3Flash := #stations.current[#i].kp8Config.flash[3],
                              btn3ColorOn1 := #stations.current[#i].kp8Config.colorOn1[3],
                              btn3ColorOn2 := #stations.current[#i].kp8Config.colorOn2[3],
                              btn3ColorOff := #stations.current[#i].kp8Config.colorOff[3],
                              btn4Activate := #stations.current[#i].kp8Config.activate[4],
                              btn4Mode := #stations.current[#i].kp8Config.mode[4],
                              btn4Group := #stations.current[#i].kp8Config.group[4],
                              btn4Flash := #stations.current[#i].kp8Config.flash[4],
                              btn4ColorOn1 := #stations.current[#i].kp8Config.colorOn1[4],
                              btn4ColorOn2 := #stations.current[#i].kp8Config.colorOn2[4],
                              btn4ColorOff := #stations.current[#i].kp8Config.colorOff[4],
                              btn5Activate := #stations.current[#i].kp8Config.activate[5],
                              btn5Mode := #stations.current[#i].kp8Config.mode[5],
                              btn5Group := #stations.current[#i].kp8Config.group[5],
                              btn5Flash := #stations.current[#i].kp8Config.flash[5],
                              btn5ColorOn1 := #stations.current[#i].kp8Config.colorOn1[5],
                              btn5ColorOn2 := #stations.current[#i].kp8Config.colorOn2[5],
                              btn5ColorOff := #stations.current[#i].kp8Config.colorOff[5],
                              btn6Activate := #stations.current[#i].kp8Config.activate[6],
                              btn6Mode := #stations.current[#i].kp8Config.mode[6],
                              btn6Group := #stations.current[#i].kp8Config.group[6],
                              btn6Flash := #stations.current[#i].kp8Config.flash[6],
                              btn6ColorOn1 := #stations.current[#i].kp8Config.colorOn1[6],
                              btn6ColorOn2 := #stations.current[#i].kp8Config.colorOn2[6],
                              btn6ColorOff := #stations.current[#i].kp8Config.colorOff[6],
                              btn7Activate := #stations.current[#i].kp8Config.activate[7],
                              btn7Mode := #stations.current[#i].kp8Config.mode[7],
                              btn7Group := #stations.current[#i].kp8Config.group[7],
                              btn7Flash := #stations.current[#i].kp8Config.flash[7],
                              btn7ColorOn1 := #stations.current[#i].kp8Config.colorOn1[7],
                              btn7ColorOn2 := #stations.current[#i].kp8Config.colorOn2[7],
                              btn7ColorOff := #stations.current[#i].kp8Config.colorOff[7],
                              btnStatesOut => #stations.current[#i].btnStates,
                              btnColorsOut => #stations.current[#i].kp8Out);
       END_FOR;
   END_REGION
END_REGION

REGION Network 5: RESET INITIALIZATION REQUESTS
   // Initialization requests are no longer necessare and are turned off to maintain program integrity.
   RUNG wire#powerrail
      #instResetInitRequest(constants := #constants, stations := #stations)
   END_RUNG
   // the same network as SCL:
   #instResetInitRequest(constants := #constants, stations := #stations);   // "Reset Init Requests"
END_REGION

REGION Network 6: BARCODE SCREEN
   RUNG wire#powerrail
      #instHMIBarcode(constants := #constants, partCall := "HMI".partCall, barcodeScreen := "HMI".barcode, stations := #stations)
   END_RUNG
   // the same network as SCL:
   #instHMIBarcode(constants := #constants,   // "HMI Barcod Screen"
                   partCall := "HMI".partCall,
                   barcodeScreen := "HMI".barcode,
                   stations := #stations);
END_REGION

REGION Network 7: PART TIMERS
   RUNG wire#powerrail
      #instPartTimers(constants := #constants, stations := #stations)
   END_RUNG
   // the same network as SCL:
   #instPartTimers(constants := #constants, stations := #stations);   // "Part Timers"
END_REGION

REGION Network 8: RECORD PART REQUEST
   RUNG wire#powerrail
      #instRecordPartRequest(pRow := "Parts".pRow, requests := "Parts".requests, stations := #stations)
   END_RUNG
   // the same network as SCL:
   #instRecordPartRequest(pRow := "Parts".pRow, requests := "Parts".requests, stations := #stations);   // "Record Part Request"
END_REGION

REGION Network 9: REMOVE PART REQUEST
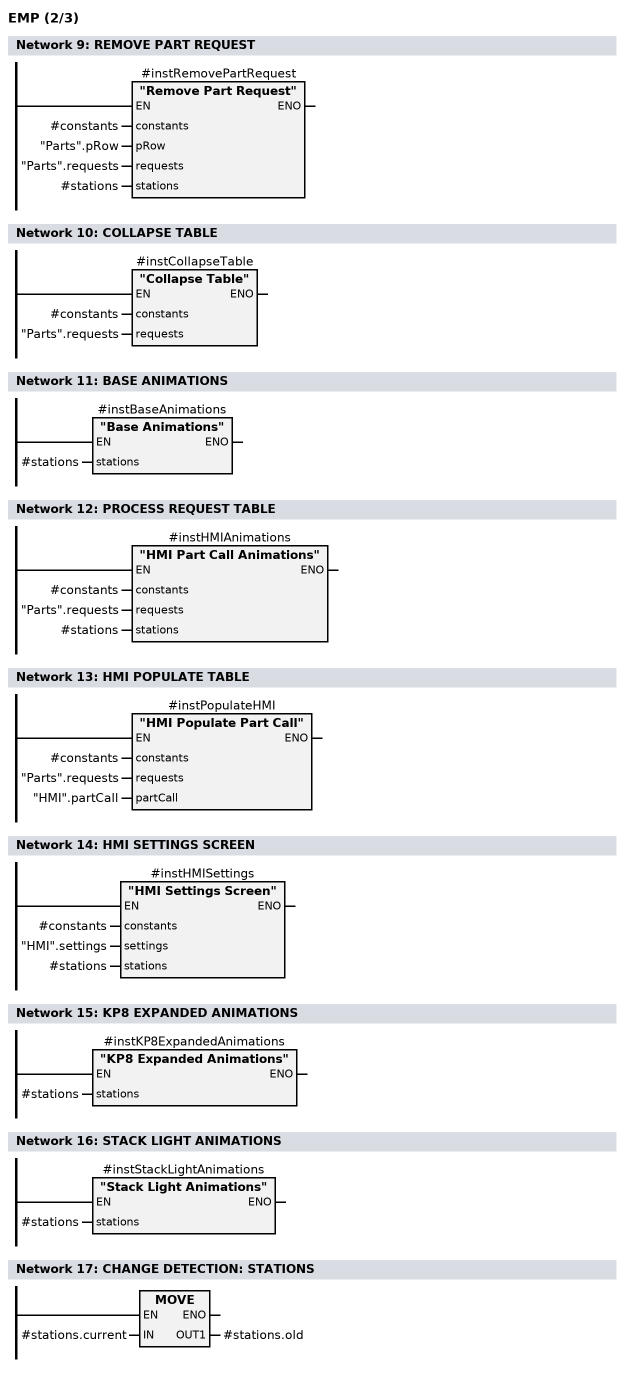
   RUNG wire#powerrail
      #instRemovePartRequest(constants := #constants, pRow := "Parts".pRow, requests := "Parts".requests, stations := #stations)
   END_RUNG
   // the same network as SCL:
   #instRemovePartRequest(constants := #constants,   // "Remove Part Request"
                          pRow := "Parts".pRow,
                          requests := "Parts".requests,
                          stations := #stations);
END_REGION

REGION Network 10: COLLAPSE TABLE
   RUNG wire#powerrail
      #instCollapseTable(constants := #constants, requests := "Parts".requests)
   END_RUNG
   // the same network as SCL:
   #instCollapseTable(constants := #constants, requests := "Parts".requests);   // "Collapse Table"
END_REGION

REGION Network 11: BASE ANIMATIONS
   RUNG wire#powerrail
      #instBaseAnimations(stations := #stations)
   END_RUNG
   // the same network as SCL:
   #instBaseAnimations(stations := #stations);   // "Base Animations"
END_REGION

REGION Network 12: PROCESS REQUEST TABLE
   RUNG wire#powerrail
      #instHMIAnimations(constants := #constants, requests := "Parts".requests, stations := #stations)
   END_RUNG
   // the same network as SCL:
   #instHMIAnimations(constants := #constants, requests := "Parts".requests, stations := #stations);   // "HMI Part Call Animations"
END_REGION

REGION Network 13: HMI POPULATE TABLE
   RUNG wire#powerrail
      #instPopulateHMI(constants := #constants, requests := "Parts".requests, partCall := "HMI".partCall)
   END_RUNG
   // the same network as SCL:
   #instPopulateHMI(constants := #constants, requests := "Parts".requests, partCall := "HMI".partCall);   // "HMI Populate Part Call"
END_REGION

REGION Network 14: HMI SETTINGS SCREEN
   RUNG wire#powerrail
      #instHMISettings(constants := #constants, settings := "HMI".settings, stations := #stations)
   END_RUNG
   // the same network as SCL:
   #instHMISettings(constants := #constants, settings := "HMI".settings, stations := #stations);   // "HMI Settings Screen"
END_REGION

REGION Network 15: KP8 EXPANDED ANIMATIONS
   RUNG wire#powerrail
      #instKP8ExpandedAnimations(stations := #stations)
   END_RUNG
   // the same network as SCL:
   #instKP8ExpandedAnimations(stations := #stations);   // "KP8 Expanded Animations"
END_REGION

REGION Network 16: STACK LIGHT ANIMATIONS
   RUNG wire#powerrail
      #instStackLightAnimations(stations := #stations)
   END_RUNG
   // the same network as SCL:
   #instStackLightAnimations(stations := #stations);   // "Stack Light Animations"
END_REGION

REGION Network 17: CHANGE DETECTION: STATIONS
   RUNG wire#powerrail
      Move(in := #stations.current, out1 => #stations.old)
   END_RUNG
   // the same network as SCL:
   #stations.old := #stations.current;
END_REGION

REGION Network 18: CHANGE DETECTION: PART CALL SCREEN
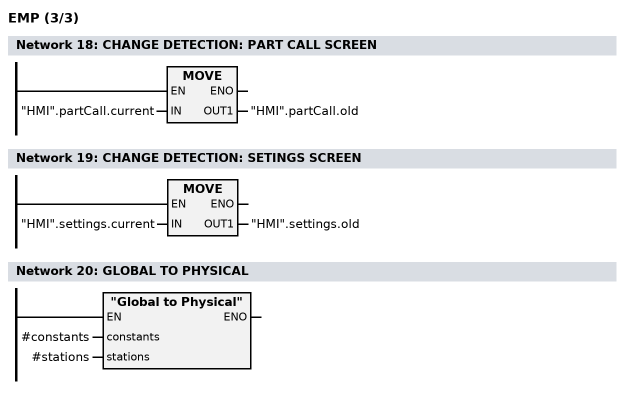
   RUNG wire#powerrail
      Move(in := "HMI".partCall.current, out1 => "HMI".partCall.old)
   END_RUNG
   // the same network as SCL:
   "HMI".partCall.old := "HMI".partCall.current;
END_REGION

REGION Network 19: CHANGE DETECTION: SETINGS SCREEN
   RUNG wire#powerrail
      Move(in := "HMI".settings.current, out1 => "HMI".settings.old)
   END_RUNG
   // the same network as SCL:
   "HMI".settings.old := "HMI".settings.current;
END_REGION

REGION Network 20: GLOBAL TO PHYSICAL
   RUNG wire#powerrail
      "Global to Physical"(constants := #constants, stations := #stations)
   END_RUNG
   // the same network as SCL:
   "Global to Physical"(constants := #constants, stations := #stations);
END_REGION
END_FUNCTION_BLOCK

FUNCTION_BLOCK "Code 128"   // FB2, SCL
{ S7_Optimized_Access := 'TRUE' }
VERSION : 0.1
   VAR_INPUT
      partNumber : String;
   END_VAR
   VAR_OUTPUT
      barcode : String;
   END_VAR
   VAR
      charsIn : Array[0..255] of Byte;
      charsOut : Array[0..255] of Byte;
      cnt : UInt;
      intVals : Array[0..255] of Int;
      sum : Int;
      checkSum : Int;
   END_VAR
   VAR_TEMP
      pn : String;
      i : Int;
   END_VAR
   VAR CONSTANT
      startChar : Char := 'Ì';
      stopChar : Char := 'Î';
   END_VAR
   // intVals[0] := 104;
BEGIN
   #pn := #partNumber;

   FOR #i := 0 TO 255 DO
       #charsIn[#i] := 16#00;
       #charsOut[#i] := 16#00;
       #intVals[#i] := 0;
   END_FOR;

   Strg_TO_Chars(Strg:=#pn,
                 pChars:=0,
                 Cnt=>#cnt,
                 Chars:=#charsIn);


   #sum := 104;
   FOR #i := 0 TO UINT_TO_INT(#cnt - 1) DO
       #intVals[#i] := CHAR_TO_INT(#charsIn[#i]) - 32;
       #intVals[#i] := #intVals[#i] * (#i + 1);
       #sum := #sum + #intVals[#i];
   END_FOR;
   #checkSum := (#sum MOD 103) + 32;
   IF #checkSum >= 127 THEN
       #checkSum := #checkSum + 68;
   END_IF;

   #charsOut[0] := #startChar;
   FOR #i := 1 TO UINT_TO_INT(#cnt) DO
       #charsOut[#i] := #charsIn[#i - 1];
   END_FOR;
   #charsOut[#cnt + 1] := INT_TO_BYTE(#checkSum);
   #charsOut[#cnt + 2] := INT_TO_BYTE(#stopChar);

   Chars_TO_Strg(Chars := #charsOut,
                 pChars := 0,
                 Cnt := #cnt + 3,
                 Strg => #barcode);
END_FUNCTION_BLOCK

FUNCTION_BLOCK "HMI Barcod Screen"   // FB3, SCL
{ S7_Optimized_Access := 'TRUE' }
VERSION : 0.1
   VAR_INPUT
      constants : "Constants";
   END_VAR
   VAR_IN_OUT
      partCall : "Part Call Screen";
      barcodeScreen : "Barcode Screen";
      stations : "Stations";
   END_VAR
   VAR
      address : UInt;
      button : UInt;
      instCode128 : "Code 128";
      codeOut : String;
      pnOut : WString[40];
      station : UInt;
      oldSelectedRow : Int;
   END_VAR
   VAR_TEMP
      orderCancelled : Int;
      processedPN : String[40];
      selectedPN : String[40];
      userOrdered : Bool;
      selectedRow : Int;
   END_VAR
   VAR CONSTANT
      maxRows : Int := 199;
   END_VAR
BEGIN
   REGION "GET USER ROW SELECTION"
       #selectedRow := "Get Part Call Row Number"(constants := #constants,
                                                  partCall := #partCall);
   END_REGION

   REGION "ON SELECTION OF A PART CALL ROW
       IF #selectedRow <> 0 THEN
           IF #selectedRow <> #oldSelectedRow THEN

               REGION "GET BUTTON AND STATION NUMBERS"
                   #address := #partCall.current[#selectedRow - 1].address;
                   "Address to Station and Button"(address := #address,
                                                   station => #station,
                                                   button => #button);
               END_REGION

               REGION "CONVERT STRING TO BARCODE"

                   REGION "COPY TO LOCALS"
                       #selectedPN := WSTRING_TO_STRING(#partCall.current[#selectedRow - 1].tfPartNumber.value);
                   END_REGION

                   REGION "CONVERT TO BARCODE"
                       #instCode128(partNumber := #processedPN,
                                    barcode => #codeOut);
                   END_REGION

                   REGION "OUTPUT FOR HMI SCREEN"
                       #barcodeScreen.partNumber := STRING_TO_WSTRING(#processedPN);
                       #barcodeScreen.barcode := #codeOut;
                   END_REGION

               END_REGION

           END_IF;
       END_IF;
   END_REGION

   REGION "PASS USER ORDERED"
       // get input
       #userOrdered := #barcodeScreen.ordered;
       // put into station
       #stations.current[#station].partOrdered[#button] := #userOrdered;
   END_REGION


   #oldSelectedRow := #selectedRow;
END_FUNCTION_BLOCK

FUNCTION_BLOCK "Initialize"   // FB4, SCL
{ S7_Optimized_Access := 'TRUE' }
VERSION : 0.1
   VAR_INPUT
      constants : "Constants";
   END_VAR
   VAR_IN_OUT
      stations : "Stations";
   END_VAR
   VAR
      rtElapsed : Real;
      rt : Struct
         elapsed : LReal;
         mem : LReal;
      END_STRUCT;
   END_VAR
   VAR_TEMP
      i : Int;
      reset : Struct
         req : Bool;
         elapsed : Real;
      END_STRUCT;
      stnCount : Int;
      init : Bool;
   END_VAR
   VAR CONSTANT
      resetLimit : Real := 1.25;
   END_VAR
BEGIN
   REGION "GET STATION COUNT"
       #stnCount := #constants.stationCount - 1;
   END_REGION

   REGION "FIRST SCAN"
       IF "FirstScan" THEN
           // initialize all stations on plc first scan
           FOR #i := 0 TO #stnCount DO
               #stations.current[#i].init.hard := TRUE;
           END_FOR;
       END_IF;
   END_REGION

   REGION "RUNTIME CALL"
       // get elapsed time
       #rt.elapsed := RUNTIME(#rt.mem);
       // convert to real data type
       #rtElapsed := LREAL_TO_REAL(#rt.elapsed);
   END_REGION

   REGION "BUTTON 0 BASED RESET TIMERS"
       FOR #i := 0 TO #stnCount DO

           REGION "PRE-CONDITION"
               // init off by default
               #init := FALSE;
               // request is button 0 on kp8
               #reset.req := #stations.current[#i].kp8In.%X0;
               // saved to shorter name
               #reset.elapsed := #stations.current[#i].elapsedTime.resetReq;
           END_REGION

           REGION "RESET REQUEST"
               IF NOT #reset.req THEN
                   #reset.elapsed := 0.0;
               END_IF;
               IF #reset.req THEN
                   // incriment elapsed time
                   #reset.elapsed := #reset.elapsed + #rtElapsed;
                   // timer expired condition
                   IF #reset.elapsed >= #resetLimit THEN
                       #init := TRUE;
                       #reset.elapsed := 0.0;
                   END_IF;
               END_IF;
               // save elapsed time
               #stations.current[#i].elapsedTime.resetReq := #reset.elapsed;
           END_REGION

           REGION "SAVE INITIALIZATIN REQUEST"
               #stations.current[#i].init.hard := #init;
           END_REGION

       END_FOR;
   END_REGION
END_FUNCTION_BLOCK

FUNCTION_BLOCK "Reset Init Requests"   // FB5, SCL
{ S7_Optimized_Access := 'TRUE' }
VERSION : 0.1
   VAR_INPUT
      constants : "Constants";
   END_VAR
   VAR_IN_OUT
      stations : "Stations";
   END_VAR
   VAR
      placeHolder : Bool;
   END_VAR
   VAR_TEMP
      i : Int;
      stnCount : Int;
   END_VAR
BEGIN
   REGION "GET STATION COUNT"
       #stnCount := #constants.stationCount - 1;
   END_REGION

   REGION "RESET INITIALIZATION REQUESTS
       FOR #i := 0 TO #stnCount DO
           #stations.current[#i].init.hard := FALSE;
           #stations.current[#i].init.soft := FALSE;
       END_FOR;
   END_REGION
END_FUNCTION_BLOCK

FUNCTION_BLOCK "Record Part Request"   // FB6, SCL
{ S7_Optimized_Access := 'TRUE' }
VERSION : 0.1
   VAR_IN_OUT
      pRow : Int;
      requests : "Part Request Data";
      stations : "Stations";
   END_VAR
   VAR
      enterAddress : Bool;
   END_VAR
   VAR_TEMP
      address : UInt;
      hasPart : Bool;
      i : Int;
      intTime : Int;
      j : Int;
      k : Int;
      logAddress : UInt;
      noPart : Bool;
      oldPartReq : Bool;
      partReq : Bool;
      partNumber : WString;
      timeTime : Time;
      wstringTime : WString;
   END_VAR
   VAR CONSTANT
      maxRows : Int := 199;
      stationCount : Int := 22;
   END_VAR
BEGIN
   REGION "MAIN LOOP"
       FOR #i := 0 TO #stationCount DO

           REGION "LOOP THROUGH BUTTONS"
               // j = 0 is excluded because it is used as a station reset button
               FOR #j := 1 TO 7 DO

                   REGION "PRE-CONDITION"
                       // bits for new request detection
                       #partReq := #stations.current[#i].btnStates[#j];
                       #oldPartReq := #stations.old[#i].btnStates[#j];
                   END_REGION

                   REGION "DETERMINE STATE"
                       // new request detection
                       IF #partReq AND NOT #oldPartReq THEN
                           // save to local
                           #partNumber := #stations.current[#i].partNumbers[#j];
                           // no part number
                           IF LEN(#partNumber) = 0 THEN
                               #hasPart := FALSE;
                               #noPart := TRUE;
                           END_IF;
                           // has part number
                           IF LEN(#partNumber) <> 0 THEN
                               #hasPart := TRUE;
                               #noPart := FALSE;
                           END_IF;
                       END_IF;
                   END_REGION

                   REGION "NO PART"
                       IF #noPart THEN
                           // turn off the lights
                           #hasPart := FALSE;
                           #noPart := FALSE;
                           #enterAddress := FALSE;
                       END_IF;
                   END_REGION

                   REGION "HAS PART"
                       IF #hasPart THEN
                           // turn off the lights
                           #hasPart := FALSE;
                           // calculate address
                           #address := (INT_TO_UINT(#i) + 1) * 10 + (INT_TO_UINT(#j) + 1);
                           // precondition enter address flag
                           #enterAddress := TRUE;
                           // check table for previous entry
                           FOR #k := 0 TO #maxRows DO
                               // save to local
                               #logAddress := #requests.row[#k].address;
                               // do not re-enter previous requests
                               IF #logAddress = #address THEN
                                   #enterAddress := FALSE;
                               END_IF;
                           END_FOR;
                       END_IF;
                   END_REGION

                   REGION "ENTER ADDRESS"
                       IF #enterAddress THEN
                           // turn off the lights
                           #enterAddress := FALSE;
                           // no processing needed
                           #requests.row[#pRow].address := #address;
                           #requests.row[#pRow].tfLine.value := #stations.current[#i].line;
                           // drop zone is unsigned so simple conversion is okay
                           #requests.row[#pRow].tfDropZone.value := USINT_TO_WSTRING(#stations.current[#i].dropZone);
                           // no processing needed
                           #requests.row[#pRow].tfPartNumber.value := #stations.current[#i].partNumbers[#j];
                           // several steps to change real to time based wstring
                           #intTime := REAL_TO_INT(#stations.current[#i].elapsedTime.partReq[#j]);
                           #timeTime := INT_TO_TIME(#intTime);
                           #wstringTime := "Time to WString"(#timeTime);
                           #requests.row[#pRow].tfTime.value := #wstringTime;
                           // incriment row pointer
                           #pRow := #pRow + 1;
                           IF #pRow > #maxRows THEN
                               #pRow := 0;
                           END_IF;
                       END_IF;
                   END_REGION

               END_FOR;
           END_REGION

       END_FOR;
   END_REGION
END_FUNCTION_BLOCK

FUNCTION_BLOCK "Part Timers"   // FB7, SCL
{ S7_Optimized_Access := 'TRUE' }
VERSION : 0.1
   VAR_INPUT
      constants : "Constants";
   END_VAR
   VAR_IN_OUT
      stations : "Stations";
   END_VAR
   VAR
      rt : "Runtime Data";
   END_VAR
   VAR_TEMP
      alottedTime : Real;
      btnCount : Int;
      elapsedTime : Real;
      i : Int;
      j : Int;
      partRequested : Bool;
      redTime : Real;
      remainingTime : Real;
      stnCount : Int;
      press : Struct
         current : Bool;
         old : Bool;
      END_STRUCT;
   END_VAR
BEGIN
   REGION "RUNTIME CALL"
       #rt.elapsed := RUNTIME(#rt.mem);
       #rt.asReal := LREAL_TO_REAL(#rt.elapsed);
   END_REGION

   REGION "GET STATION COUNT"
       #stnCount := #constants.stationCount - 1;
       #btnCount := #constants.buttonCount - 1;
   END_REGION

   REGION "MAIN LOOP"
       FOR #i := 0 TO #stnCount DO
           // j := 0 would be the reset button so it is skipped
           FOR #j := 1 TO #btnCount DO

               REGION "RESET PART TIMER"
                   #press.current := #stations.current[#i].btnStates[#j];
                   #press.old := #stations.old[#i].btnStates[#j];
                   IF NOT #press.current AND #press.old THEN
                           #stations.current[#i].elapsedTime.partReq[#j] := 0.0;
                   END_IF;
               END_REGION

               REGION "PART REQUEST TIMER"
                   // get and check button state 
                   #partRequested := #stations.current[#i].btnStates[#j];
                   IF #partRequested THEN

                       REGION "OUTPUT ELLAPSED TIME"
                           // get saved time
                           #elapsedTime := #stations.current[#i].elapsedTime.partReq[#j];
                           // add elapsed time
                           #elapsedTime := #elapsedTime + #rt.asReal;
                           // save new value
                           #stations.current[#i].elapsedTime.partReq[#j] := #elapsedTime;
                       END_REGION

                   END_IF;
               END_REGION

           END_FOR;
       END_FOR;
   END_REGION
END_FUNCTION_BLOCK

FUNCTION_BLOCK "Base Animations"   // FB8, SCL
{ S7_Optimized_Access := 'TRUE' }
VERSION : 0.1
   VAR_IN_OUT
      stations : "Stations";
   END_VAR
   VAR_TEMP
      animation : Int;
      i : Int;
      j : Int;
      partRequested : Bool;
      partOrdered : Bool;
      elapsedTime : Real;
      criticalTime : Real;
      alottedTime : Real;
      remainingTime : Real;
   END_VAR
   VAR CONSTANT
      stationCount : Int := 22;
      anDefault : USInt := 0;
      anRequested : USInt := 1;
      anSolidRed : USInt := 2;
      anFlashRed : USInt := 3;
      anPartOrdered : USInt := 4;
   END_VAR
BEGIN
   REGION "MAIN LOOP"
       FOR #i := 0 TO #stationCount DO
           // j := 0 would be the reset button so it is skipped
           FOR #j := 1 TO 7 DO

               REGION "PART REQUEST TIMER"

                   REGION "COPY TO LOCAL"
                       #partRequested := #stations.current[#i].btnStates[#j];
                       #partOrdered := #stations.current[#i].partOrdered[#j];
                   END_REGION

                   REGION "PART REQUESTED"
                       IF #partRequested THEN

                           REGION "GET LOCAL VARIABLES"
                               // remaining time
                               #elapsedTime := #stations.current[#i].elapsedTime.partReq[#j];
                               #alottedTime := #stations.current[#i].presetTime.allotted[#j];
                               #remainingTime := #alottedTime - #elapsedTime;
                               // critical time
                               #criticalTime := #stations.current[#i].presetTime.critical[#j];
                           END_REGION

                           REGION "DEFAULT ANIMATION STATE"
                               IF #remainingTime > #criticalTime THEN
                                   #animation := #anRequested;
                               END_IF;
                           END_REGION

                           REGION "SOLID RED ANIMATION STATE"
                               IF #remainingTime <= #criticalTime AND #elapsedTime > 0.0 THEN
                                   #animation := #anSolidRed;
                               END_IF;
                           END_REGION

                           REGION "FLASHING RED ANIMATION STATE
                               IF #remainingTime <= 0.0 THEN
                                   #animation := #anFlashRed;
                               END_IF;
                           END_REGION ;

                           REGION "ORDERED"
                               IF #partOrdered THEN
                                   #animation := #anPartOrdered;
                               END_IF;
                           END_REGION

                       END_IF;
                   END_REGION

                   REGION "PART NOT REQUESTED"
                       IF NOT #partRequested THEN
                           #animation := #anDefault;
                       END_IF;
                   END_REGION

                   REGION "OUTPUT"
                       #stations.current[#i].animations[#j] := #animation;
                   END_REGION

               END_REGION

           END_FOR;
       END_FOR;
   END_REGION
END_FUNCTION_BLOCK

FUNCTION_BLOCK "HMI Part Call Animations"   // FB9, SCL
{ S7_Optimized_Access := 'TRUE' }
VERSION : 0.1
   VAR_INPUT
      constants : "Constants";
   END_VAR
   VAR_IN_OUT
      requests : "Part Request Data";
      stations : "Stations";
   END_VAR
   VAR
      station : Int;
      button : Int;
   END_VAR
   VAR_TEMP
      address : Int;
      animator : UInt;
      maxRows : Int;
      timeAsReal : Real;
      timeAsTime : WString;
      i : Int;
   END_VAR
BEGIN
   REGION "COPY TO LOCAL"
       #maxRows := #constants.partReqRows - 1;
   END_REGION

   REGION "ITERATE THROUGH VISIBLE TABLE ROWS"
       FOR #i := 0 TO #maxRows DO

           REGION "COPY TO LOCAL"
               #address := UINT_TO_INT(#requests.row[#i].address);
           END_REGION

           REGION "HIDE UNPOPULATED ROWS"
               IF #address = 0 THEN
                   #requests.row[#i].pbSelection.visibility := FALSE;
                   #requests.row[#i].rtBackground.visibility := FALSE;
                   #animator := 0;
                   #requests.row[#i].tfDropZone.visibility := FALSE;
                   #requests.row[#i].tfDropZone.animator := #animator;
                   #requests.row[#i].tfLine.visibility := FALSE;
                   #requests.row[#i].tfLine.animator := #animator;
                   #requests.row[#i].tfPartNumber.visibility := FALSE;
                   #requests.row[#i].tfPartNumber.animator := #animator;
                   #requests.row[#i].tfTime.visibility := FALSE;
                   #requests.row[#i].tfTime.animator := #animator;
               END_IF;
           END_REGION

           REGION "ANIMATE POPULATED ROWS"

               REGION "ANIMATE ROWS WITH DATA"
                   IF #address <> 0 THEN

                       REGION "GET POINTERS FOR STATION ARRAY"
                           #station := #address / 10 - 1;
                           #button := #address MOD 10 - 1;
                       END_REGION

                       REGION "ANIMATIONS"

                           REGION "PUSHBUTTON VISIBILITY"
                               #requests.row[#i].pbSelection.visibility := TRUE;
                           END_REGION

                           REGION "BACKGROUND VISIBILITY"
                               #requests.row[#i].rtBackground.visibility := TRUE;
                           END_REGION

                           REGION "ANIMATOR VALUE"
                               #animator := INT_TO_UINT(#stations.current[#station].animations[#button]);
                           END_REGION

                           REGION "DROP ZONE" 
                               #requests.row[#i].tfDropZone.visibility := TRUE;
                               #requests.row[#i].tfDropZone.value := UINT_TO_WSTRING(#stations.current[#station].dropZone);
                               #requests.row[#i].tfDropZone.animator := #animator;
                           END_REGION

                           REGION "LINE"
                               #requests.row[#i].tfLine.visibility := TRUE;
                               #requests.row[#i].tfLine.value := #stations.current[#station].line;
                               #requests.row[#i].tfLine.animator := #animator;
                           END_REGION

                           REGION "PART NUMBER"
                               #requests.row[#i].tfPartNumber.visibility := TRUE;
                               #requests.row[#i].tfPartNumber.value := #stations.current[#station].partNumbers[#button];
                               #requests.row[#i].tfPartNumber.animator := #animator;
                           END_REGION

                           REGION "TIME"
                               #requests.row[#i].tfTime.visibility := TRUE;
                               #timeAsReal := #stations.current[#station].presetTime.allotted[#button];
                               #timeAsReal -= #stations.current[#station].elapsedTime.partReq[#button];
                               #requests.row[#i].tfTime.value := "Real to WString Timer"(#timeAsReal);
                               #requests.row[#i].tfTime.animator := #animator;
                           END_REGION

                       END_REGION

                   END_IF;
               END_REGION

           END_REGION

       END_FOR;
   END_REGION
END_FUNCTION_BLOCK

FUNCTION_BLOCK "KP8 Expanded Animations"   // FB10, SCL
{ S7_Optimized_Access := 'TRUE' }
VERSION : 0.1
   VAR_IN_OUT
      stations : "Stations";
   END_VAR
   VAR_TEMP
      i : Int;
      j : Int;
      colorBox : DWord;
      animation : Int;
      redMask : DWord;
   END_VAR
   VAR CONSTANT
      stationCount : Int := 22;
      buttonCount : Int := 7;
      anSolidRed : USInt := 2;
      anFlashRed : USInt := 3;
   END_VAR
BEGIN
   REGION "LOOP THROUGH STATIONS"
       FOR #i := 0 TO #stationCount DO

           REGION "LOOP THROUGH BUTTONS"
               FOR #j := 0 TO #buttonCount DO

                   REGION "GET ANIMATION"
                       #animation := #stations.current[#i].animations[#j];
                   END_REGION

                   REGION "SOLID RED"
                       IF #animation = #anSolidRed THEN
                           #colorBox := #stations.current[#i].kp8Out;
                           #redMask := 16#FEFEFE00;
                           #redMask := ROL_DWORD(IN := #redMask,
                                                 N := INT_TO_UINT(#j));
                           #colorBox := #colorBox AND #redMask;
                           #redMask := 16#100_0000;
                           #redMask := ROL_DWORD(IN := #redMask,
                                                 N := INT_TO_UINT(#j));
                           #colorBox := #colorBox OR #redMask;
                           #stations.current[#i].kp8Out := #colorBox;
                       END_IF;
                   END_REGION

                   REGION "FLASHING RED"
                       IF #animation = #anFlashRed THEN

                           REGION "RED ON"
                               IF "Clock_1Hz" THEN
                                   #colorBox := #stations.current[#i].kp8Out;
                                   #redMask := 16#FEFEFE00;
                                   #redMask := ROL_DWORD(IN := #redMask,
                                                         N := INT_TO_UINT(#j));
                                   #colorBox := #colorBox AND #redMask;
                                   #redMask := 16#100_0000;
                                   #redMask := ROL_DWORD(IN := #redMask,
                                                         N := INT_TO_UINT(#j));
                                   #colorBox := #colorBox OR #redMask;
                                   #stations.current[#i].kp8Out := #colorBox;
                               END_IF;
                           END_REGION

                           REGION "RED OFF"
                               IF NOT "Clock_1Hz" THEN
                                   #colorBox := #stations.current[#i].kp8Out;
                                   #redMask := 16#FEFEFE00;
                                   #redMask := ROL_DWORD(IN := #redMask,
                                                         N := INT_TO_UINT(#j));
                                   #colorBox := #colorBox AND #redMask;
                                   #stations.current[#i].kp8Out := #colorBox;
                               END_IF;
                           END_REGION

                       END_IF;
                   END_REGION

               END_FOR;
           END_REGION

       END_FOR;
   END_REGION
END_FUNCTION_BLOCK

FUNCTION_BLOCK "Stack Light Animations"   // FB11, SCL
{ S7_Optimized_Access := 'TRUE' }
VERSION : 0.1
   VAR_IN_OUT
      stations : "Stations";
   END_VAR
   VAR_TEMP
      animation : Int;
      i : Int;
      j : Int;
      stackLight : DWord;
   END_VAR
   VAR CONSTANT
      anDefault : USInt := 0;
      anRequested : USInt := 1;
      anSolidRed : USInt := 2;
      anFlashRed : USInt := 3;
      anPartOrdered : USInt := 4;
      buttonCount : Int := 7;
      "Part 01" : Int := 7;
      "Part 01 Green On" : DWord := 16#0400_0000;
      "Part 01 Red On" : DWord := 16#0100_0000;
      "Part 01 Yellow On" : DWord := 16#0200_0000;
      "Part 02" : Int := 3;
      "Part 02 Green On" : DWord := 16#2000_0000;
      "Part 02 Red On" : DWord := 16#0800_0000;
      "Part 02 Yellow On" : DWord := 16#1000_0000;
      "Part 03" : Int := 6;
      "Part 03 Green On" : DWord := 16#0001_0000;
      "Part 03 Red On" : DWord := 16#4000_0000;
      "Part 03 Yellow On" : DWord := 16#8000_0000;
      "Part 04" : Int := 2;
      "Part 04 Green On" : DWord := 16#0008_0000;
      "Part 04 Yellow On" : DWord := 16#0004_0000;
      "Part 04 Red On" : DWord := 16#0002_0000;
      "Part 05" : Int := 5;
      "Part 05 Green On" : DWord := 16#0040_0000;
      "Part 05 Red On" : DWord := 16#0010_0000;
      "Part 05 Yellow On" : DWord := 16#0020_0000;
      "Part 06" : Int := 1;
      "Part 06 Green On" : DWord := 16#0000_0200;
      "Part 06 Red On" : DWord := 16#0080_0000;
      "Part 06 Yellow On" : DWord := 16#0000_0100;
      stationCount : Int := 22;
   END_VAR
BEGIN
   REGION "LOOP THROUGH STATIONS"
       FOR #i := 0 TO #stationCount DO

           REGION "LOOP THROUGH BUTTONS"
               FOR #j := 0 TO #buttonCount DO

                   REGION "COPY INTO LOCAL"
                       #stackLight := #stations.current[#i].stackLightOut;
                       #animation := #stations.current[#i].animations[#j];
                   END_REGION

                   REGION "GREEN"
                       IF #animation = #anDefault THEN
                           CASE #j OF
                               #"Part 01":
                                   #stackLight := #stackLight AND (NOT #"Part 01 Red On");
                                   #stackLight := #stackLight AND (NOT #"Part 01 Yellow On");
                                   #stackLight := #stackLight OR #"Part 01 Green On";
                               #"Part 02":
                                   #stackLight := #stackLight AND (NOT #"Part 02 Red On");
                                   #stackLight := #stackLight AND (NOT #"Part 02 Yellow On");
                                   #stackLight := #stackLight OR #"Part 02 Green On";
                               #"Part 03":
                                   #stackLight := #stackLight AND (NOT #"Part 03 Red On");
                                   #stackLight := #stackLight AND (NOT #"Part 03 Yellow On");
                                   #stackLight := #stackLight OR #"Part 03 Green On";
                               #"Part 04":
                                   #stackLight := #stackLight AND (NOT #"Part 04 Red On");
                                   #stackLight := #stackLight AND (NOT #"Part 04 Yellow On");
                                   #stackLight := #stackLight OR #"Part 04 Green On";
                               #"Part 05":
                                   #stackLight := #stackLight AND (NOT #"Part 05 Red On");
                                   #stackLight := #stackLight AND (NOT #"Part 05 Yellow On");
                                   #stackLight := #stackLight OR #"Part 05 Green On";
                               #"Part 06":
                                   #stackLight := #stackLight AND (NOT #"Part 06 Red On");
                                   #stackLight := #stackLight AND (NOT #"Part 06 Yellow On");
                                   #stackLight := #stackLight OR #"Part 06 Green On";
                               ELSE
                                   ;
                           END_CASE;
                       END_IF;
                   END_REGION

                   REGION "YELLOW"
                       IF #animation = #anRequested THEN
                           CASE #j OF
                               #"Part 01":
                                   #stackLight := #stackLight AND (NOT #"Part 01 Red On");
                                   #stackLight := #stackLight OR #"Part 01 Yellow On";
                                   #stackLight := #stackLight AND (NOT #"Part 01 Green On");
                               #"Part 02":
                                   #stackLight := #stackLight AND (NOT #"Part 02 Red On");
                                   #stackLight := #stackLight OR #"Part 02 Yellow On";
                                   #stackLight := #stackLight AND (NOT #"Part 02 Green On");
                               #"Part 03":
                                   #stackLight := #stackLight AND (NOT #"Part 03 Red On");
                                   #stackLight := #stackLight OR #"Part 03 Yellow On";
                                   #stackLight := #stackLight AND (NOT #"Part 03 Green On");
                               #"Part 04":
                                   #stackLight := #stackLight AND (NOT #"Part 04 Red On");
                                   #stackLight := #stackLight OR #"Part 04 Yellow On";
                                   #stackLight := #stackLight AND (NOT #"Part 04 Green On");
                               #"Part 05":
                                   #stackLight := #stackLight AND (NOT #"Part 05 Red On");
                                   #stackLight := #stackLight OR #"Part 05 Yellow On";
                                   #stackLight := #stackLight AND (NOT #"Part 05 Green On");
                               #"Part 06":
                                   #stackLight := #stackLight AND (NOT #"Part 06 Red On");
                                   #stackLight := #stackLight OR #"Part 06 Yellow On";
                                   #stackLight := #stackLight AND (NOT #"Part 06 Green On");
                               ELSE
                                   ;
                           END_CASE;
                       END_IF;
                   END_REGION

                   REGION "SOLID RED"
                       IF #animation = #anSolidRed THEN
                           CASE #j OF
                               #"Part 01":
                                   #stackLight := #stackLight OR #"Part 01 Red On";
                                   #stackLight := #stackLight AND (NOT #"Part 01 Yellow On");
                                   #stackLight := #stackLight AND (NOT #"Part 01 Green On");
                               #"Part 02":
                                   #stackLight := #stackLight OR #"Part 02 Red On";
                                   #stackLight := #stackLight AND (NOT #"Part 02 Yellow On");
                                   #stackLight := #stackLight AND (NOT #"Part 02 Green On");
                               #"Part 03":
                                   #stackLight := #stackLight OR #"Part 03 Red On";
                                   #stackLight := #stackLight AND (NOT #"Part 03 Yellow On");
                                   #stackLight := #stackLight AND (NOT #"Part 03 Green On");
                               #"Part 04":
                                   #stackLight := #stackLight OR #"Part 04 Red On";
                                   #stackLight := #stackLight AND (NOT #"Part 04 Yellow On");
                                   #stackLight := #stackLight AND (NOT #"Part 04 Green On");
                               #"Part 05":
                                   #stackLight := #stackLight OR #"Part 05 Red On";
                                   #stackLight := #stackLight AND (NOT #"Part 05 Yellow On");
                                   #stackLight := #stackLight AND (NOT #"Part 05 Green On");
                               #"Part 06":
                                   #stackLight := #stackLight OR #"Part 06 Red On";
                                   #stackLight := #stackLight AND (NOT #"Part 06 Yellow On");
                                   #stackLight := #stackLight AND (NOT #"Part 06 Green On");
                               ELSE
                                   ;
                           END_CASE;
                       END_IF;
                   END_REGION

                   REGION "FLASHING RED"
                       IF #animation = #anFlashRed THEN

                           REGION "RED ON"
                               IF "Clock_1Hz" THEN
                                   CASE #j OF
                                       #"Part 01":
                                           #stackLight := #stackLight OR #"Part 01 Red On";
                                           #stackLight := #stackLight AND (NOT #"Part 01 Yellow On");
                                           #stackLight := #stackLight AND (NOT #"Part 01 Green On");
                                       #"Part 02":
                                           #stackLight := #stackLight OR #"Part 02 Red On";
                                           #stackLight := #stackLight AND (NOT #"Part 02 Yellow On");
                                           #stackLight := #stackLight AND (NOT #"Part 02 Green On");
                                       #"Part 03":
                                           #stackLight := #stackLight OR #"Part 03 Red On";
                                           #stackLight := #stackLight AND (NOT #"Part 03 Yellow On");
                                           #stackLight := #stackLight AND (NOT #"Part 03 Green On");
                                       #"Part 04":
                                           #stackLight := #stackLight OR #"Part 04 Red On";
                                           #stackLight := #stackLight AND (NOT #"Part 04 Yellow On");
                                           #stackLight := #stackLight AND (NOT #"Part 04 Green On");
                                       #"Part 05":
                                           #stackLight := #stackLight OR #"Part 05 Red On";
                                           #stackLight := #stackLight AND (NOT #"Part 05 Yellow On");
                                           #stackLight := #stackLight AND (NOT #"Part 05 Green On");
                                       #"Part 06":
                                           #stackLight := #stackLight OR #"Part 06 Red On";
                                           #stackLight := #stackLight AND (NOT #"Part 06 Yellow On");
                                           #stackLight := #stackLight AND (NOT #"Part 06 Green On");
                                       ELSE
                                           ;
                                   END_CASE;
                               END_IF;
                           END_REGION

                           REGION "RED OFF"
                               IF NOT "Clock_1Hz" THEN
                                   CASE #j OF
                                       #"Part 01":
                                           #stackLight := #stackLight AND (NOT #"Part 01 Red On");
                                           #stackLight := #stackLight AND (NOT #"Part 01 Yellow On");
                                           #stackLight := #stackLight AND (NOT #"Part 01 Green On");
                                       #"Part 02":
                                           #stackLight := #stackLight AND (NOT #"Part 02 Red On");
                                           #stackLight := #stackLight AND (NOT #"Part 02 Yellow On");
                                           #stackLight := #stackLight AND (NOT #"Part 02 Green On");
                                       #"Part 03":
                                           #stackLight := #stackLight AND (NOT #"Part 03 Red On");
                                           #stackLight := #stackLight AND (NOT #"Part 03 Yellow On");
                                           #stackLight := #stackLight AND (NOT #"Part 03 Green On");
                                       #"Part 04":
                                           #stackLight := #stackLight AND (NOT #"Part 04 Red On");
                                           #stackLight := #stackLight AND (NOT #"Part 04 Yellow On");
                                           #stackLight := #stackLight AND (NOT #"Part 04 Green On");
                                       #"Part 05":
                                           #stackLight := #stackLight AND (NOT #"Part 05 Red On");
                                           #stackLight := #stackLight AND (NOT #"Part 05 Yellow On");
                                           #stackLight := #stackLight AND (NOT #"Part 05 Green On");
                                       #"Part 06":
                                           #stackLight := #stackLight AND (NOT #"Part 06 Red On");
                                           #stackLight := #stackLight AND (NOT #"Part 06 Yellow On");
                                           #stackLight := #stackLight AND (NOT #"Part 06 Green On");
                                       ELSE
                                           ;
                                   END_CASE;
                               END_IF;
                           END_REGION

                       END_IF;
                   END_REGION

                   REGION "COPY OUT TO GLOBAL"
                       #stations.current[#i].stackLightOut := #stackLight;
                   END_REGION

               END_FOR;
           END_REGION

       END_FOR;
   END_REGION
END_FUNCTION_BLOCK

FUNCTION_BLOCK "KP8 Button Activation"   // FB12, SCL
{ S7_Optimized_Access := 'TRUE' }
VERSION : 0.1
   VAR_INPUT
      constants : "Constants";
   END_VAR
   VAR_IN_OUT
      stations : "Stations";
   END_VAR
   VAR_TEMP
      btnCount : Int;
      currentPNs : Array[0..7] of WString[40];
      i : Int;
      init : Bool;
      j : Int;
      stnCount : Int;
      temp : Int;
   END_VAR
BEGIN
   REGION "GET STATION COUNT"
       #stnCount := #constants.stationCount - 1;
       #btnCount := #constants.buttonCount - 1;
   END_REGION

   REGION "LOOP THROUGH STATIONS"
       FOR #i := 0 TO #stnCount DO

           #currentPNs := #stations.current[#i].partNumbers;

           REGION "LOOP THROUGH BUTTONS"
               FOR #j := 0 TO #btnCount DO

                       REGION "ACTIVATE BUTTON"
                           IF LEN(#currentPNs[#j]) <> 0 THEN
                               #stations.current[#i].kp8Config.activate[#j] := TRUE;
                               #stations.current[#i].kp8Config.colorOff[#j] := 'green';
                               #stations.current[#i].kp8Config.colorOn1[#j] := 'yellow';
                               #stations.current[#i].kp8Config.colorOn2[#j] := '';
                               #stations.current[#i].kp8Config.flash[#j] := FALSE;
                               #stations.current[#i].kp8Config.group[#j] := 0;
                               #stations.current[#i].kp8Config.mode[#j] := TRUE;
                           END_IF;
                       END_REGION

                       REGION "DEACTIVATE BUTTON"
                           IF LEN(#currentPNs[#j]) = 0 THEN
                               #stations.current[#i].kp8Config.activate[#j] := FALSE;
                               #stations.current[#i].kp8Config.colorOff[#j] := '';
                               #stations.current[#i].kp8Config.colorOn1[#j] := '';
                               #stations.current[#i].kp8Config.colorOn2[#j] := '';
                               #stations.current[#i].kp8Config.flash[#j] := FALSE;
                               #stations.current[#i].kp8Config.group[#j] := 0;
                               #stations.current[#i].kp8Config.mode[#j] := FALSE;
                           END_IF;
                       END_REGION

               END_FOR;
           END_REGION

           REGION "SOFT INIT"
               IF #stations.current[#i].kp8Config <> #stations.old[#i].kp8Config THEN
                   #stations.current[#i].init.soft := TRUE;
               END_IF;
           END_REGION

       END_FOR;
   END_REGION
END_FUNCTION_BLOCK

FUNCTION_BLOCK "Remove Part Request"   // FB13, SCL
{ S7_Optimized_Access := 'TRUE' }
VERSION : 0.1
   VAR_INPUT
      constants : "Constants";
   END_VAR
   VAR_IN_OUT
      pRow : Int;
      requests : "Part Request Data";
      stations : "Stations";
   END_VAR
   VAR_TEMP
      address : UInt;
      blankRow : "Table Row";
      hasPart : Bool;
      i : Int;
      j : Int;
      k : Int;
      logAddress : UInt;
      maxRows : Int;
      noPart : Bool;
      oldPartReq : Bool;
      partNumber : WString;
      partReq : Bool;
      pRemoveRow : Int;
      removeAddress : Bool;
   END_VAR
   VAR CONSTANT
      buttonCount : Int := 7;
      stationCount : Int := 22;
   END_VAR
BEGIN
   #maxRows := #constants.partReqRows - 1;

   REGION "LOOP THROUGH STATIONS"
       FOR #i := 0 TO #stationCount DO

           REGION "LOOP THROUGH BUTTONS"
               FOR #j := 1 TO #buttonCount DO

                   REGION "PRE-CONDITION"
                       // copy bits for falling edge detection
                       #partReq := #stations.current[#i].btnStates[#j];
                       #oldPartReq := #stations.old[#i].btnStates[#j];
                   END_REGION

                   REGION "DETERMINE STATE"
                       // falling edge detection
                       IF NOT #partReq AND #oldPartReq THEN
                           // copy to local
                           #partNumber := #stations.current[#i].partNumbers[#j];
                           // no part
                           IF #partNumber = wstring#'' THEN
                               #hasPart := FALSE;
                               #noPart := TRUE;
                           END_IF;
                           // has part
                           IF #partNumber <> wstring#'' THEN
                               #hasPart := TRUE;
                               #noPart := FALSE;
                           END_IF;
                       END_IF;
                   END_REGION

                   REGION "NO PART"
                       IF #noPart THEN
                           // turn off the lights
                           #hasPart := FALSE;
                           #noPart := FALSE;
                       END_IF;

                   END_REGION

                   REGION "HAS PART"
                       IF #hasPart THEN
                           // turn off the lights
                           #hasPart := FALSE;
                           // calculate address
                           #address := (INT_TO_UINT(#i) + 1) * 10 + (INT_TO_UINT(#j) + 1);
                           // precondition remove address flag
                           #removeAddress := FALSE;
                           // check table for previous entry
                           FOR #k := 0 TO #maxRows DO
                               #logAddress := #requests.row[#k].address;
                               // remove matching address flag
                               IF #logAddress = #address THEN
                                   #removeAddress := TRUE;
                                   #pRemoveRow := #k;
                               END_IF;
                           END_FOR;
                       END_IF;
                   END_REGION

                   REGION "REMOVE ADDRESS"
                       IF #removeAddress THEN

                           // turn off the lights
                           #removeAddress := FALSE;

                           REGION "REMOVAL PROCESS"
                               #requests.row[#pRemoveRow] := #blankRow;
                           END_REGION

                           REGION "ADJUST TABLE BLANK ROW POINTER"
                               // decriment row pointer
                               #pRow := #pRow - 1;
                               IF #pRow < 0 THEN
                                   #pRow := 0;
                               END_IF;
                           END_REGION

                       END_IF;
                   END_REGION

               END_FOR;

           END_REGION

       END_FOR;
   END_REGION
END_FUNCTION_BLOCK

FUNCTION_BLOCK "HMI Settings Screen"   // FB14, LAD
{ S7_Optimized_Access := 'TRUE' }
VERSION : 0.1
   VAR_INPUT
      constants : "Constants";
   END_VAR
   VAR_IN_OUT
      settings : "Settings Screen";
      stations : "Stations";
   END_VAR
   VAR
      btnSlctCount : Int;
      btnNumber : Int;
      evalSlct : Bool;
      firstStation : Int := 0;
      stnSlctCount : Int;
      tmrSelAllStn : TON_TIME;
      tmrDeslctAllStn : TON_TIME;
      tmrSelAllBtn : TON_TIME;
      tmrDeslctAllBtn : TON_TIME;
      tmrTimeOut : TON_TIME;
   END_VAR
   VAR_TEMP
      btnSelected : Bool;
      count : Int;
      currentBtn : Bool;
      i : Int;
      j : Int;
      partNumber : WString;
      newEntry : Bool;
      oldBtn : Bool;
      oldCount : Int;
      oldPN : WString;
      oldStnNumber : Int;
      pBtn : Int;
      pSN : Int;
      stnSelected : Bool;
      stnNumber : Int;
      timerWString : WString;
      timerReal : Real;
      viewStn : Int;
   END_VAR
   VAR CONSTANT
      adjBtnCount : Int := 6;
      adjStnCount : Int := 23;
      buttonCount : Int := 5;
      stationCount : Int := 22;
      msPerSec : Real := 1000.0;
      ptSelectAll : Time := T#1S500MS;
      ptTimeOut : Time := t#5M;
   END_VAR
BEGIN

REGION Network 1: CLEAR PART NUMBER WHEN MODE DESELECTED
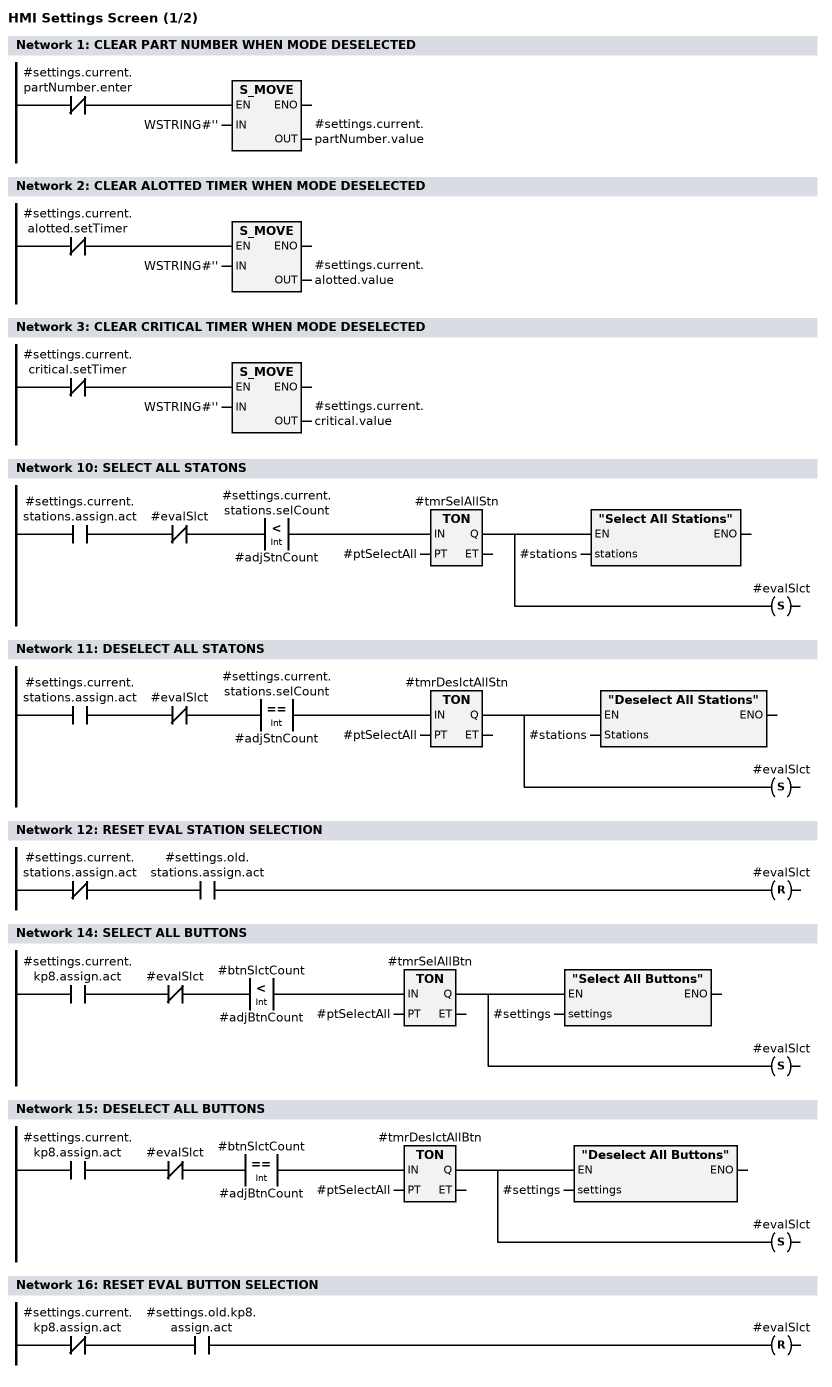
   RUNG wire#powerrail
      I_Contact( #settings.current.partNumber.enter )
      S_Move(in := WSTRING#'', out => #settings.current.partNumber.value)
   END_RUNG
   // the same network as SCL:
   IF NOT #settings.current.partNumber.enter THEN #settings.current.partNumber.value := WSTRING#''; END_IF;
END_REGION

REGION Network 2: CLEAR ALOTTED TIMER WHEN MODE DESELECTED
   RUNG wire#powerrail
      I_Contact( #settings.current.alotted.setTimer )
      S_Move(in := WSTRING#'', out => #settings.current.alotted.value)
   END_RUNG
   // the same network as SCL:
   IF NOT #settings.current.alotted.setTimer THEN #settings.current.alotted.value := WSTRING#''; END_IF;
END_REGION

REGION Network 3: CLEAR CRITICAL TIMER WHEN MODE DESELECTED
   RUNG wire#powerrail
      I_Contact( #settings.current.critical.setTimer )
      S_Move(in := WSTRING#'', out => #settings.current.critical.value)
   END_RUNG
   // the same network as SCL:
   IF NOT #settings.current.critical.setTimer THEN #settings.current.critical.value := WSTRING#''; END_IF;
END_REGION

REGION Network 5 (SCL): COUNT SELECTED STATIONS
   #count := 0;
   FOR #i := 0 TO #stationCount DO
       #stnSelected := #stations.current[#i].settings.selected;
       IF #stnSelected THEN
           #count += 1;
       END_IF;
   END_FOR;
   #settings.current.stations.selCount := #count;
END_REGION

REGION Network 6 (SCL): POPULATE STATION NUMBER FOR SINGLE OR ALL STATIONS
   #count := #settings.current.stations.selCount;
   #oldCount := #settings.old.stations.selCount;
   IF #count <> #oldCount
       AND (#count = 1 OR #count = #stationCount + 1) THEN
           FOR #i := 0 TO #stationCount DO
               #stnSelected := #stations.current[#i].settings.selected;
               IF #stnSelected THEN
                   #stnNumber := #i + 1;
                   #settings.current.viewingStation.number := #stnNumber;
                   EXIT;
               END_IF;
           END_FOR;
   END_IF;
END_REGION

REGION Network 7 (SCL): VIEW NEXT STATION IF STATION REMOVED FROM SELECTION
   #count := #settings.current.stations.selCount;
   #oldCount := #settings.old.stations.selCount;
   IF #count <> #oldCount THEN
       #stnNumber := #settings.current.viewingStation.number;
       #pSN := #stnNumber - 1;
       #stnSelected := #stations.current[#pSN].settings.selected;
       IF NOT #stnSelected THEN
           FOR #i := #stnNumber + 1 TO #stationCount DO
               #stnSelected := #stations.current[#i].settings.selected;
               IF #stnSelected THEN
                   #stnNumber := #i + 1;
                   #settings.current.viewingStation.number := #stnNumber;
                   EXIT;
               END_IF;
           END_FOR;
       END_IF;
   END_IF;
END_REGION

REGION Network 8 (SCL): PREVIOUS STATION
   #count := #settings.current.stations.selCount;
   IF #count <> 0 THEN
       #currentBtn := #settings.current.viewingStation.previous.act;
       #oldBtn := #settings.old.viewingStation.previous.act;
       IF #currentBtn AND NOT #oldBtn THEN
           #i := #settings.current.viewingStation.number - 2;
           IF #i > #stationCount THEN
               #i := #stationCount;
           END_IF;
           #stnSelected := #stations.current[#i].settings.selected;
           WHILE NOT #stnSelected DO
               #i := #i - 1;
               IF #i < 0 THEN
                   #i := #stationCount;
               END_IF;
               #stnSelected := #stations.current[#i].settings.selected;
           END_WHILE;
           #settings.current.viewingStation.number := #i + 1;
       END_IF;
   END_IF;
END_REGION

REGION Network 9 (SCL): NEXT STATION
   #count := #settings.current.stations.selCount;
   IF #count <> 0 THEN
       #currentBtn := #settings.current.viewingStation.next.act;
       #oldBtn := #settings.old.viewingStation.next.act;
       IF #currentBtn AND NOT #oldBtn THEN
           #viewStn := #settings.current.viewingStation.number;
           IF #viewStn > #stationCount THEN
               #viewStn := 0;
           END_IF;
           #stnSelected := #stations.current[#viewStn].settings.selected;
           WHILE NOT #stnSelected DO
               #viewStn += 1;
               IF #viewStn > #stationCount THEN
                   #viewStn := 0;
               END_IF;
               #stnSelected := #stations.current[#viewStn].settings.selected;
           END_WHILE;
           #viewStn += 1;
           #settings.current.viewingStation.number := #viewStn;
       END_IF;
   END_IF;
END_REGION

REGION Network 10: SELECT ALL STATONS
   #tmrSelAllStn(IN := #settings.current.stations.assign.act AND NOT #evalSlct AND (#settings.current.stations.selCount < #adjStnCount),   // TON
                 PT := #ptSelectAll);
   IF #tmrSelAllStn.Q THEN
       "Select All Stations"(stations := #stations);
       #evalSlct := TRUE;
   END_IF;
END_REGION

REGION Network 11: DESELECT ALL STATONS
   #tmrDeslctAllStn(IN := #settings.current.stations.assign.act AND NOT #evalSlct AND (#settings.current.stations.selCount = #adjStnCount),   // TON
                    PT := #ptSelectAll);
   IF #tmrDeslctAllStn.Q THEN
       "Deselect All Stations"(Stations := #stations);
       #evalSlct := TRUE;
   END_IF;
END_REGION

REGION Network 12: RESET EVAL STATION SELECTION
   RUNG wire#powerrail
      I_Contact( #settings.current.stations.assign.act )
      Contact( #settings.old.stations.assign.act )
      R_Coil( #evalSlct )
   END_RUNG
   // the same network as SCL:
   IF NOT #settings.current.stations.assign.act AND #settings.old.stations.assign.act THEN
       #evalSlct := FALSE;
   END_IF;
END_REGION

